C05456=1029.880,242.416,382.549,170.287,45.519,158.700
C05457=1029.874,242.168,382.577,170.284,45.520,158.700
C05458=1029.867,241.920,382.606,170.281,45.521,158.700
C05459=1029.860,241.672,382.634,170.277,45.522,158.700
C05460=1029.854,241.423,382.662,170.274,45.524,158.700
C05461=1029.847,241.175,382.691,170.271,45.524,158.699
C05462=1029.841,240.926,382.719,170.267,45.525,158.699
C05463=1029.834,240.678,382.748,170.264,45.527,158.699
C05464=1029.828,240.429,382.776,170.261,45.527,158.699
C05465=1029.821,240.181,382.805,170.259,45.529,158.699
C05466=1029.814,239.933,382.832,170.254,45.530,158.699
C05467=1029.808,239.685,382.861,170.252,45.531,158.699
C05468=1029.801,239.436,382.889,170.249,45.532,158.699
C05469=1029.794,239.189,382.918,170.245,45.533,158.699
C05470=1029.788,238.940,382.945,170.242,45.535,158.699
C05471=1029.781,238.692,382.974,170.239,45.535,158.698
C05472=1029.775,238.444,383.002,170.235,45.537,158.698
C05473=1029.768,238.195,383.030,170.232,45.538,158.698
C05474=1029.761,237.947,383.058,170.229,45.539,158.698
C05475=1029.754,237.698,383.087,170.225,45.540,158.698
C05476=1029.748,237.449,383.115,170.223,45.541,158.698
C05477=1029.741,237.202,383.143,170.220,45.543,158.698
C05478=1029.734,236.953,383.171,170.216,45.543,158.698
C05479=1029.727,236.705,383.199,170.213,45.545,158.698
C05480=1029.722,236.456,383.227,170.210,45.546,158.698
C05481=1029.715,236.208,383.255,170.207,45.547,158.698
C05482=1029.708,235.960,383.283,170.203,45.548,158.697
C05483=1029.701,235.711,383.311,170.200,45.549,158.697
C05484=1029.694,235.463,383.339,170.198,45.550,158.697
C05485=1029.687,235.215,383.367,170.194,45.552,158.697
C05486=1029.678,234.842,383.409,170.189,45.554,158.697
C05487=1029.668,234.468,383.450,170.184,45.556,158.697
C05488=1029.658,234.095,383.493,170.181,45.557,158.697
C05489=1029.649,233.721,383.535,170.176,45.559,158.697
C05490=1029.642,233.473,383.563,170.172,45.560,158.697
C05491=1029.635,233.225,383.591,170.169,45.561,158.697
C05492=1029.629,232.976,383.618,170.166,45.563,158.697
C05493=1029.622,232.728,383.646,170.163,45.563,158.696
C05494=1029.615,232.480,383.675,170.159,45.565,158.696
C05495=1029.608,232.231,383.702,170.157,45.566,158.696
C05496=1029.602,231.983,383.731,170.154,45.567,158.696
C05497=1029.596,231.734,383.758,170.151,45.568,158.696
C05498=1029.589,231.486,383.786,170.147,45.570,158.696
C05499=1029.582,231.237,383.814,170.144,45.571,158.696
C05500=1029.576,230.989,383.842,170.141,45.572,158.696
C05501=1029.570,230.741,383.869,170.138,45.573,158.696
C05502=1029.563,230.493,383.897,170.135,45.575,158.696
C05503=1029.556,230.244,383.924,170.132,45.576,158.696
C05504=1029.550,229.996,383.952,170.129,45.577,158.696
C05505=1029.543,229.747,383.980,170.126,45.578,158.696
C05506=1029.536,229.499,384.008,170.122,45.580,158.696
C05507=1029.530,229.250,384.035,170.120,45.581,158.696
C05508=1029.523,229.002,384.063,170.117,45.583,158.696
C05509=1029.516,228.754,384.091,170.114,45.583,158.695
C05510=1029.509,228.505,384.118,170.110,45.585,158.695
C05511=1029.503,228.257,384.146,170.107,45.586,158.695
C05512=1029.497,228.008,384.173,170.104,45.588,158.695
C05513=1029.490,227.760,384.201,170.102,45.589,158.695
C05514=1029.484,227.511,384.228,170.098,45.590,158.695
C05515=1029.477,227.263,384.256,170.095,45.591,158.695
C05516=1029.470,227.015,384.284,170.092,45.593,158.695
C05517=1029.463,226.766,384.311,170.089,45.594,158.695
C05518=1029.457,226.518,384.338,170.085,45.596,158.695
C05519=1029.450,226.270,384.365,170.083,45.597,158.695
C05520=1029.444,226.021,384.393,170.080,45.598,158.695
C05521=1029.436,225.773,384.420,170.077,45.600,158.695
C05522=1029.430,225.524,384.447,170.073,45.601,158.695
C05523=1029.423,225.276,384.475,170.071,45.603,158.695
C05524=1029.417,225.028,384.502,170.068,45.604,158.695
C05525=1029.410,224.779,384.529,170.065,45.605,158.695
C05526=1029.403,224.531,384.556,170.061,45.607,158.695
C05527=1029.397,224.282,384.584,170.059,45.608,158.695
C05528=1029.390,224.033,384.611,170.056,45.610,158.695
C05529=1029.383,223.785,384.638,170.053,45.611,158.695
C05530=1029.377,223.537,384.666,170.049,45.612,158.695
C05531=1029.370,223.288,384.693,170.046,45.614,158.695
C05532=1029.364,223.040,384.720,170.043,45.615,158.694
C05533=1029.356,222.792,384.748,170.041,45.616,158.694
C05534=1029.351,222.543,384.774,170.038,45.617,158.694
C05535=1029.344,222.295,384.802,170.034,45.619,158.694
C05536=1029.338,222.046,384.829,170.031,45.620,158.694
C05537=1029.330,221.798,384.856,170.029,45.621,158.694
C05538=1029.323,221.549,384.884,170.026,45.623,158.694
C05539=1029.318,221.301,384.910,170.023,45.624,158.694
C05540=1029.311,221.052,384.938,170.019,45.626,158.694
C05541=1029.304,220.804,384.965,170.016,45.627,158.694
C05542=1029.294,220.423,385.006,170.012,45.630,158.694
C05543=1029.284,220.042,385.049,170.007,45.631,158.694
C05544=1029.274,219.661,385.090,170.004,45.634,158.694
C05545=1029.264,219.279,385.131,169.999,45.636,158.694
C05546=1029.257,219.032,385.158,169.995,45.638,158.694
C05547=1029.251,218.783,385.185,169.993,45.639,158.694
C05548=1029.244,218.534,385.212,169.990,45.640,158.694
C05549=1029.237,218.286,385.239,169.987,45.642,158.694
C05550=1029.230,218.038,385.265,169.984,45.643,158.694
C05551=1029.224,217.789,385.293,169.980,45.645,158.694
C05552=1029.217,217.540,385.319,169.978,45.647,158.694
C05553=1029.211,217.292,385.346,169.975,45.648,158.694
C05554=1029.203,217.044,385.373,169.972,45.649,158.694
C05555=1029.197,216.795,385.400,169.970,45.651,158.694
C05556=1029.191,216.547,385.426,169.966,45.652,158.694
C05557=1029.183,216.298,385.453,169.963,45.654,158.694
C05558=1029.177,216.050,385.480,169.961,45.656,158.694
C05559=1029.170,215.802,385.507,169.958,45.657,158.694
C05560=1029.164,215.552,385.534,169.955,45.658,158.694
C05561=1029.156,215.304,385.561,169.951,45.660,158.694
C05562=1029.151,215.056,385.587,169.948,45.661,158.694
C05563=1029.144,214.807,385.614,169.946,45.663,158.694
C05564=1029.137,214.558,385.641,169.943,45.665,158.694
C05565=1029.131,214.310,385.667,169.940,45.666,158.694
C05566=1029.124,214.062,385.695,169.938,45.667,158.694
C05567=1029.117,213.813,385.721,169.934,45.669,158.694
C05568=1029.110,213.565,385.747,169.931,45.671,158.694
C05569=1029.104,213.316,385.774,169.929,45.672,158.694
C05570=1029.098,213.068,385.800,169.926,45.674,158.694
C05571=1029.091,212.819,385.828,169.923,45.675,158.694
C05572=1029.084,212.571,385.854,169.920,45.676,158.694
C05573=1029.078,212.322,385.881,169.917,45.679,158.694
C05574=1029.071,212.073,385.907,169.914,45.680,158.694
C05575=1029.065,211.825,385.934,169.911,45.681,158.694
C05576=1029.058,211.576,385.960,169.908,45.683,158.694
C05577=1029.051,211.328,385.987,169.906,45.685,158.695
C05578=1029.045,211.080,386.014,169.903,45.686,158.695
C05579=1029.038,210.831,386.041,169.900,45.687,158.695
C05580=1029.032,210.583,386.067,169.897,45.689,158.694
C05581=1029.025,210.334,386.094,169.894,45.691,158.695
C05582=1029.018,210.086,386.120,169.891,45.692,158.695
C05583=1029.011,209.837,386.146,169.889,45.694,158.695
C05584=1029.005,209.589,386.173,169.886,45.696,158.695
C05585=1028.998,209.340,386.199,169.883,45.697,158.695
C05586=1028.991,209.091,386.226,169.881,45.698,158.695
C05587=1028.985,208.843,386.252,169.877,45.701,158.695
C05588=1028.978,208.594,386.279,169.874,45.702,158.695
C05589=1028.972,208.346,386.305,169.872,45.703,158.695
C05590=1028.965,208.097,386.331,169.869,45.705,158.695
C05591=1028.958,207.849,386.357,169.866,45.707,158.695
C05592=1028.951,207.601,386.384,169.864,45.708,158.695
C05593=1028.946,207.352,386.410,169.861,45.710,158.695
C05594=1028.938,207.103,386.436,169.857,45.712,158.695
C05595=1028.932,206.855,386.462,169.855,45.714,158.695
C05596=1028.925,206.606,386.488,169.852,45.715,158.695
C05597=1028.918,206.358,386.514,169.849,45.716,158.695
C05598=1028.908,205.982,386.554,169.845,45.720,158.695
C05599=1028.899,205.606,386.594,169.840,45.722,158.695
C05600=1028.888,205.231,386.633,169.837,45.724,158.695
C05601=1028.878,204.855,386.673,169.832,45.727,158.695
C05602=1028.852,203.809,386.777,169.464,45.624,158.634
C05603=1028.846,203.560,386.802,169.460,45.626,158.634
C05604=1028.841,203.311,386.826,169.456,45.628,158.634
C05605=1028.835,203.063,386.851,169.452,45.631,158.634
C05606=1028.829,202.814,386.876,169.449,45.633,158.634
C05607=1028.822,202.566,386.900,169.444,45.636,158.634
C05608=1028.817,202.317,386.925,169.441,45.638,158.635
C05609=1028.811,202.069,386.950,169.437,45.641,158.635
C05610=1028.805,201.819,386.975,169.433,45.643,158.635
C05611=1028.799,201.570,386.999,169.430,45.646,158.635
C05612=1028.793,201.322,387.024,169.426,45.648,158.635
C05613=1028.787,201.073,387.048,169.423,45.650,158.635
C05614=1028.781,200.825,387.073,169.418,45.653,158.635
C05615=1028.775,200.576,387.098,169.415,45.656,158.635
C05616=1028.769,200.327,387.122,169.411,45.658,158.635
C05617=1028.763,200.078,387.146,169.407,45.660,158.635
C05618=1028.757,199.830,387.171,169.403,45.663,158.636
C05619=1028.751,199.581,387.195,169.400,45.666,158.636
C05620=1028.745,199.332,387.220,169.395,45.668,158.636
C05621=1028.739,199.083,387.244,169.392,45.671,158.636
C05622=1028.733,198.834,387.268,169.389,45.673,158.636
C05623=1028.727,198.585,387.292,169.384,45.676,158.636
C05624=1028.721,198.338,387.317,169.381,45.679,158.636
C05625=1028.714,198.089,387.341,169.377,45.682,158.637
C05626=1028.709,197.839,387.366,169.374,45.684,158.637
C05627=1028.703,197.591,387.389,169.370,45.687,158.637
C05628=1028.697,197.342,387.414,169.366,45.689,158.637
C05629=1028.691,197.093,387.438,169.363,45.692,158.637
C05630=1028.685,196.844,387.462,169.358,45.695,158.637
C05631=1028.679,196.596,387.486,169.355,45.697,158.637
C05632=1028.672,196.347,387.510,169.352,45.700,158.637
C05633=1028.667,196.098,387.534,169.348,45.703,158.638
C05634=1028.660,195.849,387.558,169.344,45.705,158.638
C05635=1028.655,195.601,387.582,169.340,45.707,158.638
C05636=1028.648,195.352,387.606,169.337,45.710,158.638
C05637=1028.643,195.103,387.631,169.333,45.712,158.638
C05638=1028.636,194.854,387.655,169.329,45.716,158.638
C05639=1028.631,194.606,387.679,169.326,45.718,158.638
C05640=1028.624,194.357,387.703,169.322,45.721,158.639
C05641=1028.619,194.108,387.727,169.319,45.723,158.639
C05642=1028.612,193.859,387.751,169.315,45.726,158.639
C05643=1028.606,193.611,387.775,169.311,45.729,158.639
C05644=1028.601,193.362,387.799,169.308,45.731,158.639
C05645=1028.594,193.113,387.823,169.305,45.734,158.639
C05646=1028.589,192.865,387.847,169.301,45.736,158.640
C05647=1028.582,192.616,387.871,169.297,45.740,158.640
C05648=1028.577,192.366,387.895,169.293,45.742,158.640
C05649=1028.571,192.117,387.919,169.290,45.745,158.640
C05650=1028.565,191.869,387.943,169.286,45.747,158.640
C05651=1028.559,191.621,387.967,169.283,45.750,158.640
C05652=1028.553,191.372,387.991,169.279,45.752,158.640
C05653=1028.548,191.123,388.015,169.275,45.755,158.641
C05654=1028.542,190.874,388.038,169.272,45.758,158.641
C05655=1028.536,190.625,388.063,169.269,45.760,158.641
C05656=1028.530,190.377,388.086,169.265,45.763,158.641
C05657=1028.523,190.128,388.111,169.261,45.766,158.641
C05658=1028.518,189.879,388.135,169.258,45.769,158.641
C05659=1028.512,189.630,388.158,169.254,45.771,158.641
C05660=1028.506,189.381,388.182,169.251,45.774,158.642
C05661=1028.500,189.133,388.206,169.247,45.776,158.642
C05662=1028.495,188.884,388.230,169.244,45.779,158.642
C05663=1028.488,188.600,388.257,169.240,45.782,158.642
C05664=1028.482,188.317,388.284,169.235,45.785,158.642
C05665=1028.474,188.034,388.311,169.232,45.788,158.643
C05666=1028.468,187.751,388.338,169.228,45.791,158.643
C05667=1028.463,187.502,388.362,169.224,45.794,158.643
C05668=1028.456,187.253,388.386,169.221,45.797,158.643
C05669=1028.450,187.005,388.410,169.218,45.799,158.643
C05670=1028.445,186.756,388.433,169.213,45.802,158.643
C05671=1028.439,186.507,388.457,169.210,45.804,158.643
C05672=1028.434,186.257,388.481,169.207,45.807,158.644
C05673=1028.428,186.009,388.504,169.203,45.810,158.644
C05674=1028.422,185.761,388.528,169.200,45.812,158.644
C05675=1028.417,185.512,388.552,169.197,45.815,158.644
C05676=1028.410,185.263,388.576,169.193,45.817,158.644
C05677=1028.405,185.014,388.599,169.190,45.820,158.644
C05678=1028.399,184.765,388.623,169.186,45.823,158.645
C05679=1028.393,184.517,388.647,169.183,45.826,158.645
C05680=1028.388,184.268,388.670,169.180,45.829,158.645
C05681=1028.381,184.019,388.694,169.176,45.831,158.645
C05682=1028.376,183.770,388.718,169.172,45.834,158.645
C05683=1028.370,183.521,388.741,169.168,45.836,158.645
C05684=1028.364,183.272,388.764,169.165,45.839,158.646
C05685=1028.359,183.024,388.789,169.162,45.842,158.646
C05686=1028.353,182.775,388.811,169.158,45.844,158.646
C05687=1028.347,182.526,388.835,169.155,45.847,158.646
C05688=1028.341,182.277,388.858,169.152,45.850,158.646
C05689=1028.335,182.028,388.881,169.149,45.853,158.647
C05690=1028.329,181.780,388.904,169.145,45.856,158.647
C05691=1028.323,181.530,388.927,169.141,45.859,158.647
C05692=1028.317,181.282,388.951,169.138,45.862,158.647
C05693=1028.311,181.033,388.974,169.135,45.865,158.647
C05694=1028.304,180.784,388.996,169.131,45.868,158.648
C05695=1028.298,180.535,389.019,169.128,45.871,158.648
C05696=1028.292,180.286,389.043,169.125,45.874,158.648
C05697=1028.286,180.037,389.066,169.121,45.876,158.648
C05698=1028.280,179.789,389.089,169.118,45.879,158.648
C05699=1028.274,179.540,389.111,169.114,45.882,158.649
C05700=1028.268,179.290,389.135,169.111,45.885,158.649
C05701=1028.262,179.041,389.157,169.107,45.888,158.649
C05702=1028.256,178.793,389.180,169.104,45.891,158.649
C05703=1028.250,178.544,389.204,169.101,45.894,158.650
C05704=1028.244,178.296,389.226,169.098,45.897,158.650
C05705=1028.238,178.047,389.249,169.094,45.900,158.650
C05706=1028.232,177.797,389.273,169.091,45.903,158.650
C05707=1028.226,177.548,389.296,169.088,45.906,158.650
C05708=1028.219,177.300,389.318,169.085,45.908,158.651
C05709=1028.214,177.051,389.341,169.080,45.912,158.651
C05710=1028.208,176.802,389.364,169.077,45.915,158.651
C05711=1028.202,176.553,389.387,169.074,45.917,158.651
C05712=1028.197,176.304,389.410,169.071,45.920,158.652
C05713=1028.190,176.056,389.432,169.067,45.923,158.652
C05714=1028.184,175.807,389.455,169.064,45.926,158.652
C05715=1028.178,175.557,389.478,169.061,45.929,158.652
C05716=1028.172,175.308,389.501,169.058,45.932,158.652
C05717=1028.166,175.060,389.524,169.054,45.934,158.653
C05718=1028.160,174.811,389.547,169.051,45.937,158.653
C05719=1028.154,174.562,389.570,169.048,45.940,158.653
C05720=1028.149,174.313,389.593,169.044,45.943,158.653
C05721=1028.142,174.064,389.615,169.041,45.946,158.653
C05722=1028.136,173.815,389.638,169.038,45.949,158.654
C05723=1028.131,173.566,389.661,169.035,45.952,158.654
C05724=1028.125,173.318,389.684,169.031,45.955,158.654
C05725=1028.118,173.069,389.706,169.028,45.958,158.654
C05726=1028.113,172.820,389.729,169.025,45.961,158.655
C05727=1028.106,172.536,389.755,169.021,45.965,158.655
C05728=1028.099,172.253,389.781,169.018,45.968,158.655
C05729=1028.093,171.969,389.807,169.013,45.971,158.655
C05730=1028.086,171.685,389.832,169.009,45.975,158.656
C05731=1028.080,171.436,389.855,169.006,45.978,158.656
C05732=1028.074,171.187,389.878,169.003,45.980,158.656
C05733=1028.068,170.939,389.901,169.001,45.983,158.656
C05734=1028.063,170.690,389.923,168.997,45.986,158.657
C05735=1028.057,170.441,389.945,168.994,45.989,158.657
C05736=1028.052,170.192,389.968,168.991,45.992,158.657
C05737=1028.045,169.943,389.991,168.988,45.995,158.657
C05738=1028.039,169.695,390.014,168.984,45.998,158.658
C05739=1028.034,169.446,390.037,168.981,46.001,158.658
C05740=1028.028,169.196,390.059,168.978,46.004,158.658
C05741=1028.022,168.948,390.081,168.975,46.007,158.658
C05742=1028.016,168.699,390.104,168.971,46.010,158.658
C05743=1028.010,168.450,390.127,168.968,46.013,158.659
C05744=1028.004,168.201,390.149,168.965,46.015,158.659
C05745=1027.998,167.952,390.172,168.961,46.018,158.659
C05746=1027.993,167.703,390.195,168.958,46.021,158.659
C05747=1027.987,167.454,390.218,168.955,46.024,158.659
C05748=1027.981,167.205,390.239,168.952,46.027,158.660
C05749=1027.976,166.956,390.262,168.948,46.030,158.660
C05750=1027.970,166.708,390.285,168.945,46.032,158.660
C05751=1027.964,166.458,390.307,168.942,46.035,158.660
C05752=1027.958,166.209,390.329,168.940,46.038,158.661
C05753=1027.952,165.961,390.352,168.936,46.041,158.661
C05754=1027.947,165.711,390.375,168.933,46.044,158.661
C05755=1027.941,165.463,390.396,168.930,46.047,158.661
C05756=1027.935,165.214,390.419,168.927,46.050,158.662
C05757=1027.930,164.965,390.442,168.923,46.053,158.662
C05758=1027.924,164.716,390.465,168.920,46.056,158.662
C05759=1027.918,164.467,390.486,168.917,46.059,158.662
C05760=1027.912,164.218,390.509,168.914,46.062,158.662
C05761=1027.907,163.970,390.532,168.911,46.064,158.663
C05762=1027.901,163.720,390.553,168.908,46.067,158.663
C05763=1027.895,163.471,390.576,168.905,46.070,158.663
C05764=1027.890,163.222,390.599,168.902,46.073,158.663
C05765=1027.884,162.973,390.622,168.898,46.076,158.664
C05766=1027.878,162.725,390.644,168.895,46.079,158.664
C05767=1027.873,162.476,390.666,168.892,46.082,158.664
C05768=1027.867,162.227,390.689,168.890,46.085,158.664
C05769=1027.861,161.978,390.710,168.887,46.088,158.665
C05770=1027.856,161.729,390.733,168.883,46.091,158.665
C05771=1027.850,161.480,390.755,168.880,46.094,158.665
C05772=1027.844,161.231,390.777,168.877,46.097,158.665
C05773=1027.838,160.982,390.800,168.874,46.100,158.665
C05774=1027.833,160.734,390.822,168.870,46.103,158.666
C05775=1027.828,160.484,390.845,168.868,46.105,158.666
C05776=1027.821,160.235,390.867,168.865,46.108,158.666
C05777=1027.816,159.986,390.889,168.862,46.111,158.666
C05778=1027.811,159.737,390.911,168.858,46.114,158.667
C05779=1027.805,159.488,390.933,168.855,46.117,158.667
C05780=1027.799,159.239,390.956,168.853,46.120,158.667
C05781=1027.793,158.990,390.977,168.850,46.123,158.668
C05782=1027.787,158.742,390.999,168.847,46.126,158.668
C05783=1027.782,158.492,391.021,168.843,46.129,158.668
C05784=1027.776,158.243,391.043,168.840,46.132,158.668
C05785=1027.769,157.994,391.065,168.837,46.135,158.668
C05786=1027.764,157.746,391.087,168.834,46.139,158.669
C05787=1027.758,157.497,391.109,168.831,46.142,158.669
C05788=1027.752,157.247,391.131,168.827,46.145,158.669
C05789=1027.746,156.998,391.152,168.825,46.147,158.670
C05790=1027.740,156.750,391.173,168.822,46.151,158.670
C05791=1027.733,156.465,391.199,168.818,46.154,158.670
C05792=1027.726,156.182,391.224,168.815,46.158,158.670
C05793=1027.720,155.897,391.248,168.811,46.162,158.671
C05794=1027.713,155.614,391.273,168.808,46.165,158.671
C05795=1027.708,155.364,391.295,168.805,46.168,158.671
C05796=1027.702,155.115,391.317,168.802,46.171,158.672
C05797=1027.696,154.866,391.339,168.799,46.174,158.672
C05798=1027.690,154.618,391.361,168.796,46.177,158.672
C05799=1027.684,154.369,391.383,168.793,46.180,158.672
C05800=1027.678,154.119,391.405,168.790,46.184,158.673
C05801=1027.673,153.871,391.426,168.787,46.187,158.673
C05802=1027.666,153.622,391.447,168.784,46.190,158.673
C05803=1027.661,153.372,391.470,168.780,46.192,158.673
C05804=1027.655,153.124,391.491,168.778,46.196,158.674
C05805=1027.649,152.874,391.513,168.775,46.199,158.674
C05806=1027.643,152.625,391.534,168.772,46.202,158.674
C05807=1027.638,152.377,391.555,168.769,46.205,158.675
C05808=1027.631,152.128,391.577,168.766,46.208,158.675
C05809=1027.625,151.878,391.599,168.762,46.211,158.675
C05810=1027.620,151.630,391.620,168.760,46.214,158.675
C05811=1027.613,151.381,391.642,168.757,46.218,158.676
C05812=1027.607,151.131,391.663,168.754,46.221,158.676
C05813=1027.603,150.883,391.685,168.751,46.224,158.676
C05814=1027.596,150.633,391.707,168.748,46.227,158.677
C05815=1027.591,150.385,391.728,168.745,46.230,158.677
C05816=1027.585,150.136,391.750,168.742,46.233,158.677
C05817=1027.578,149.887,391.771,168.739,46.236,158.677
C05818=1027.573,149.637,391.792,168.736,46.240,158.678
C05819=1027.567,149.388,391.813,168.733,46.243,158.678
C05820=1027.561,149.140,391.835,168.730,46.246,158.678
C05821=1027.555,148.890,391.856,168.728,46.249,158.679
C05822=1027.549,148.641,391.878,168.724,46.252,158.679
C05823=1027.544,148.393,391.899,168.721,46.255,158.679
C05824=1027.537,148.144,391.921,168.718,46.258,158.679
C05825=1027.532,147.895,391.942,168.715,46.261,158.680
C05826=1027.526,147.645,391.963,168.713,46.264,158.680
C05827=1027.520,147.397,391.984,168.710,46.267,158.680
C05828=1027.514,147.148,392.006,168.707,46.271,158.681
C05829=1027.508,146.898,392.028,168.703,46.274,158.681
C05830=1027.503,146.650,392.049,168.700,46.277,158.681
C05831=1027.497,146.400,392.070,168.698,46.280,158.681
C05832=1027.491,146.151,392.091,168.695,46.283,158.682
C05833=1027.485,145.902,392.113,168.692,46.286,158.682
C05834=1027.480,145.653,392.133,168.689,46.290,158.682
C05835=1027.474,145.404,392.155,168.686,46.293,158.682
C05836=1027.468,145.155,392.176,168.684,46.296,158.683
C05837=1027.461,144.906,392.197,168.680,46.299,158.683
C05838=1027.455,144.657,392.218,168.677,46.303,158.683
C05839=1027.450,144.408,392.239,168.674,46.306,158.684
C05840=1027.444,144.158,392.260,168.671,46.309,158.684
C05841=1027.438,143.910,392.282,168.669,46.312,158.684
C05842=1027.432,143.661,392.303,168.666,46.315,158.685
C05843=1027.426,143.412,392.323,168.663,46.319,158.685
C05844=1027.420,143.163,392.345,168.660,46.322,158.685
C05845=1027.414,142.914,392.366,168.657,46.324,158.685
C05846=1027.409,142.664,392.387,168.654,46.328,158.686
C05847=1027.403,142.416,392.408,168.651,46.331,158.686
C05848=1027.396,142.166,392.429,168.648,46.335,158.686
C05849=1027.391,141.918,392.450,168.646,46.337,158.687
C05850=1027.385,141.668,392.471,168.643,46.340,158.687
C05851=1027.379,141.419,392.492,168.640,46.344,158.687
C05852=1027.373,141.170,392.514,168.637,46.347,158.688
C05853=1027.368,140.921,392.534,168.633,46.350,158.688
C05854=1027.362,140.673,392.555,168.631,46.353,158.688
C05855=1027.355,140.388,392.579,168.627,46.357,158.688
C05856=1027.349,140.103,392.603,168.625,46.361,158.689
C05857=1027.342,139.819,392.627,168.621,46.364,158.689
C05858=1027.335,139.535,392.651,168.618,46.368,158.689
C05859=1027.330,139.286,392.672,168.615,46.371,158.690
C05860=1027.323,139.037,392.693,168.612,46.374,158.690
C05861=1027.318,138.788,392.713,168.609,46.377,158.690
C05862=1027.312,138.539,392.735,168.607,46.381,158.691
C05863=1027.306,138.290,392.755,168.604,46.384,158.691
C05864=1027.300,138.040,392.776,168.601,46.387,158.691
C05865=1027.294,137.792,392.797,168.598,46.390,158.692
C05866=1027.288,137.543,392.817,168.596,46.394,158.692
C05867=1027.282,137.294,392.839,168.592,46.397,158.692
C05868=1027.277,137.044,392.859,168.589,46.400,158.693
C05869=1027.270,136.795,392.880,168.587,46.403,158.693
C05870=1027.265,136.546,392.901,168.584,46.407,158.693
C05871=1027.259,136.297,392.921,168.581,46.410,158.693
C05872=1027.253,136.048,392.942,168.578,46.413,158.694
C05873=1027.247,135.799,392.963,168.576,46.416,158.694
C05874=1027.241,135.550,392.983,168.573,46.420,158.694
C05875=1027.235,135.301,393.004,168.570,46.423,158.695
C05876=1027.229,135.052,393.025,168.567,46.426,158.695
C05877=1027.223,134.803,393.046,168.565,46.429,158.695
C05878=1027.217,134.554,393.065,168.561,46.432,158.696
C05879=1027.211,134.304,393.086,168.558,46.436,158.696
C05880=1027.206,134.056,393.108,168.555,46.439,158.696
C05881=1027.200,133.807,393.128,168.553,46.442,158.697
C05882=1027.194,133.557,393.149,168.550,46.445,158.697
C05883=1027.188,133.308,393.169,168.547,46.449,158.697
C05884=1027.182,133.060,393.190,168.545,46.452,158.697
C05885=1027.176,132.810,393.210,168.542,46.455,158.698
C05886=1027.171,132.561,393.231,168.539,46.458,158.698
C05887=1027.165,132.312,393.251,168.536,46.462,158.698
C05888=1027.159,132.062,393.272,168.534,46.465,158.699
C05889=1027.152,131.814,393.292,168.531,46.468,158.699
C05890=1027.147,131.565,393.313,168.527,46.471,158.699
C05891=1027.141,131.315,393.334,168.525,46.475,158.700
C05892=1027.135,131.066,393.354,168.522,46.478,158.700
C05893=1027.130,130.817,393.374,168.519,46.482,158.700
C05894=1027.124,130.568,393.394,168.517,46.484,158.701
C05895=1027.118,130.319,393.415,168.514,46.488,158.701
C05896=1027.112,130.070,393.436,168.511,46.491,158.701
C05897=1027.106,129.822,393.456,168.508,46.495,158.702
C05898=1027.099,129.572,393.476,168.506,46.497,158.702
C05899=1027.093,129.323,393.496,168.503,46.501,158.702
C05900=1027.088,129.074,393.517,168.500,46.505,158.703
C05901=1027.082,128.825,393.537,168.497,46.508,158.703
C05902=1027.076,128.575,393.556,168.495,46.511,158.703
C05903=1027.070,128.326,393.576,168.492,46.515,158.704
C05904=1027.063,128.077,393.596,168.489,46.518,158.704
C05905=1027.058,127.828,393.617,168.486,46.521,158.704
C05906=1027.052,127.579,393.637,168.484,46.525,158.705
C05907=1027.045,127.329,393.657,168.480,46.528,158.705
C05908=1027.039,127.081,393.677,168.478,46.532,158.705
C05909=1027.034,126.831,393.698,168.475,46.534,158.705
C05910=1027.028,126.583,393.718,168.472,46.538,158.706
C05911=1027.022,126.333,393.738,168.469,46.542,158.706
C05912=1027.016,126.084,393.758,168.466,46.545,158.706
C05913=1027.010,125.835,393.778,168.464,46.548,158.707
C05914=1027.004,125.587,393.798,168.461,46.552,158.707
C05915=1026.998,125.336,393.818,168.458,46.555,158.707
C05916=1026.992,125.087,393.838,168.456,46.558,158.708
C05917=1026.986,124.839,393.858,168.453,46.561,158.708
C05918=1026.980,124.590,393.878,168.450,46.565,158.708
C05919=1026.974,124.305,393.901,168.447,46.569,158.709
C05920=1026.966,124.021,393.924,168.444,46.572,158.709
C05921=1026.959,123.736,393.947,168.441,46.576,158.710
C05922=1026.953,123.452,393.970,168.437,46.580,158.710
C05923=1026.947,123.203,393.990,168.435,46.583,158.710
C05924=1026.941,122.954,394.010,168.432,46.587,158.711
C05925=1026.935,122.704,394.029,168.429,46.590,158.711
C05926=1026.929,122.455,394.050,168.427,46.593,158.711
C05927=1026.923,122.206,394.070,168.424,46.596,158.712
C05928=1026.917,121.957,394.090,168.421,46.600,158.712
C05929=1026.911,121.708,394.110,168.419,46.603,158.712
C05930=1026.906,121.459,394.129,168.416,46.607,158.713
C05931=1026.900,121.209,394.150,168.413,46.610,158.713
C05932=1026.894,120.960,394.170,168.411,46.613,158.713
C05933=1026.888,120.711,394.190,168.408,46.617,158.714
C05934=1026.882,120.462,394.209,168.405,46.620,158.714
C05935=1026.876,120.213,394.229,168.403,46.623,158.714
C05936=1026.870,119.964,394.249,168.400,46.626,158.714
C05937=1026.864,119.715,394.270,168.398,46.630,158.715
C05938=1026.859,119.465,394.289,168.395,46.633,158.715
C05939=1026.853,119.216,394.309,168.391,46.636,158.715
C05940=1026.847,118.968,394.329,168.390,46.640,158.716
C05941=1026.841,118.718,394.348,168.386,46.643,158.716
C05942=1026.835,118.469,394.368,168.383,46.647,158.716
C05943=1026.830,118.220,394.389,168.381,46.649,158.717
C05944=1026.824,117.971,394.408,168.378,46.653,158.717
C05945=1026.818,117.722,394.428,168.375,46.656,158.717
C05946=1026.811,117.472,394.449,168.373,46.659,158.718
C05947=1026.806,117.223,394.468,168.370,46.663,158.718
C05948=1026.800,116.974,394.488,168.368,46.666,158.718
C05949=1026.795,116.725,394.508,168.365,46.670,158.719
C05950=1026.789,116.476,394.528,168.362,46.673,158.719
C05951=1026.783,116.227,394.547,168.360,46.676,158.719
C05952=1026.777,115.978,394.567,168.357,46.679,158.720
C05953=1026.771,115.729,394.587,168.355,46.683,158.720
C05954=1026.765,115.480,394.607,168.352,46.686,158.720
C05955=1026.759,115.230,394.626,168.349,46.689,158.721
C05956=1026.754,114.981,394.646,168.346,46.692,158.721
C05957=1026.749,114.732,394.666,168.344,46.696,158.721
C05958=1026.743,114.483,394.686,168.341,46.698,158.722
C05959=1026.737,114.234,394.706,168.338,46.702,158.722
C05960=1026.731,113.985,394.725,168.336,46.705,158.722
C05961=1026.725,113.736,394.745,168.333,46.709,158.723
C05962=1026.720,113.486,394.765,168.330,46.712,158.723
C05963=1026.713,113.237,394.785,168.328,46.715,158.723
C05964=1026.708,112.987,394.804,168.325,46.718,158.723
C05965=1026.702,112.738,394.824,168.323,46.722,158.724
C05966=1026.696,112.489,394.843,168.320,46.725,158.724
C05967=1026.690,112.240,394.863,168.317,46.728,158.724
C05968=1026.684,111.991,394.883,168.315,46.732,158.725
C05969=1026.678,111.742,394.901,168.312,46.735,158.725
C05970=1026.672,111.493,394.921,168.309,46.738,158.725
C05971=1026.666,111.243,394.940,168.307,46.742,158.726
C05972=1026.660,110.995,394.960,168.304,46.745,158.726
C05973=1026.654,110.745,394.980,168.302,46.748,158.727
C05974=1026.649,110.496,394.999,168.299,46.752,158.727
C05975=1026.643,110.247,395.019,168.296,46.755,158.727
C05976=1026.637,109.997,395.038,168.294,46.759,158.728
C05977=1026.631,109.748,395.057,168.291,46.762,158.728
C05978=1026.625,109.499,395.077,168.288,46.765,158.728
C05979=1026.619,109.250,395.096,168.286,46.769,158.729
C05980=1026.613,109.001,395.115,168.283,46.772,158.729
C05981=1026.607,108.751,395.134,168.281,46.775,158.729
C05982=1026.601,108.503,395.154,168.278,46.779,158.730
C05983=1026.594,108.218,395.176,168.275,46.783,158.730
C05984=1026.588,107.933,395.197,168.272,46.787,158.730
C05985=1026.580,107.649,395.219,168.268,46.791,158.731
C05986=1026.573,107.364,395.241,168.265,46.795,158.731
C05987=1026.567,107.115,395.261,168.263,46.798,158.732
C05988=1026.562,106.865,395.280,168.260,46.801,158.732
C05989=1026.555,106.616,395.299,168.257,46.805,158.732
C05990=1026.550,106.367,395.318,168.255,46.808,158.733
C05991=1026.544,106.118,395.338,168.252,46.811,158.733
C05992=1026.537,105.869,395.356,168.250,46.815,158.733
C05993=1026.532,105.620,395.375,168.247,46.819,158.734
C05994=1026.526,105.371,395.395,168.244,46.822,158.734
C05995=1026.520,105.122,395.413,168.242,46.825,158.734
C05996=1026.514,104.872,395.432,168.239,46.829,158.735
C05997=1026.508,104.623,395.452,168.237,46.832,158.735
C05998=1026.503,104.374,395.472,168.234,46.835,158.735
C05999=1026.496,104.125,395.490,168.231,46.839,158.736
C06000=1026.490,103.875,395.510,168.229,46.842,158.736
C06001=1026.485,103.626,395.529,168.226,46.846,158.736
C06002=1026.478,103.377,395.547,168.224,46.849,158.737
C06003=1026.473,103.127,395.567,168.221,46.852,158.737
C06004=1026.467,102.878,395.586,168.218,46.856,158.737
C06005=1026.461,102.629,395.605,168.216,46.859,158.738
C06006=1026.455,102.381,395.624,168.213,46.862,158.738
C06007=1026.449,102.131,395.643,168.211,46.866,158.738
C06008=1026.443,101.882,395.662,168.208,46.869,158.739
C06009=1026.437,101.633,395.681,168.206,46.872,158.739
C06010=1026.432,101.383,395.701,168.203,46.876,158.739
C06011=1026.425,101.134,395.719,168.200,46.879,158.739
C06012=1026.420,100.885,395.738,168.198,46.882,158.740
C06013=1026.414,100.636,395.757,168.195,46.886,158.740
C06014=1026.408,100.387,395.776,168.193,46.889,158.741
C06015=1026.402,100.138,395.795,168.190,46.893,158.741
C06016=1026.397,99.888,395.814,168.188,46.896,158.741
C06017=1026.390,99.639,395.833,168.185,46.899,158.742
C06018=1026.385,99.390,395.852,168.182,46.903,158.742
C06019=1026.378,99.140,395.871,168.180,46.906,158.742
C06020=1026.372,98.891,395.890,168.177,46.910,158.743
C06021=1026.366,98.641,395.908,168.175,46.913,158.743
C06022=1026.361,98.393,395.926,168.172,46.917,158.743
C06023=1026.355,98.143,395.946,168.169,46.920,158.744
C06024=1026.348,97.894,395.964,168.167,46.924,158.744
C06025=1026.342,97.645,395.983,168.164,46.927,158.744
C06026=1026.336,97.396,396.002,168.161,46.931,158.745
C06027=1026.330,97.147,396.021,168.159,46.934,158.745
C06028=1026.325,96.897,396.039,168.156,46.937,158.745
C06029=1026.319,96.648,396.058,168.154,46.941,158.746
C06030=1026.312,96.399,396.076,168.151,46.944,158.746
C06031=1026.307,96.150,396.096,168.148,46.948,158.746
C06032=1026.300,95.900,396.114,168.146,46.951,158.747
C06033=1026.294,95.651,396.133,168.143,46.955,158.747
C06034=1026.289,95.402,396.151,168.141,46.958,158.748
C06035=1026.282,95.153,396.170,168.138,46.962,158.748
C06036=1026.277,94.903,396.189,168.135,46.965,158.748
C06037=1026.270,94.654,396.208,168.133,46.968,158.749
C06038=1026.264,94.405,396.226,168.130,46.972,158.749
C06039=1026.259,94.156,396.244,168.128,46.975,158.749
C06040=1026.253,93.907,396.263,168.125,46.979,158.750
C06041=1026.247,93.657,396.282,168.123,46.982,158.750
C06042=1026.241,93.408,396.300,168.120,46.985,158.750
C06043=1026.235,93.159,396.319,168.117,46.989,158.750
C06044=1026.229,92.910,396.338,168.115,46.992,158.751
C06045=1026.223,92.661,396.356,168.112,46.996,158.751
C06046=1026.217,92.411,396.374,168.110,46.999,158.752
C06047=1026.211,92.127,396.396,168.107,47.003,158.752
C06048=1026.204,91.843,396.417,168.105,47.007,158.752
C06049=1026.197,91.557,396.438,168.102,47.011,158.753
C06050=1026.190,91.273,396.459,168.099,47.014,158.753
C06051=1026.184,91.024,396.478,168.096,47.018,158.754
C06052=1026.179,90.775,396.497,168.093,47.021,158.754
C06053=1026.172,90.525,396.515,168.091,47.025,158.754
C06054=1026.167,90.276,396.534,168.088,47.028,158.755
C06055=1026.161,90.026,396.552,168.086,47.031,158.755
C06056=1026.155,89.778,396.570,168.083,47.035,158.755
C06057=1026.149,89.528,396.589,168.081,47.039,158.756
C06058=1026.143,89.279,396.607,168.078,47.042,158.756
C06059=1026.137,89.030,396.626,168.075,47.045,158.756
C06060=1026.131,88.781,396.644,168.073,47.049,158.757
C06061=1026.125,88.531,396.662,168.070,47.053,158.757
C06062=1026.119,88.282,396.680,168.068,47.056,158.757
C06063=1026.113,88.033,396.698,168.065,47.059,158.758
C06064=1026.107,87.783,396.716,168.062,47.063,158.758
C06065=1026.100,87.534,396.735,168.060,47.066,158.758
C06066=1026.094,87.285,396.753,168.057,47.070,158.759
C06067=1026.089,87.036,396.772,168.055,47.074,158.759
C06068=1026.083,86.786,396.790,168.052,47.077,158.759
C06069=1026.076,86.537,396.808,168.049,47.080,158.760
C06070=1026.071,86.288,396.826,168.047,47.084,158.760
C06071=1026.064,86.039,396.845,168.045,47.088,158.760
C06072=1026.058,85.789,396.863,168.042,47.090,158.761
C06073=1026.053,85.540,396.880,168.039,47.094,158.761
C06074=1026.046,85.291,396.899,168.037,47.098,158.761
C06075=1026.040,85.041,396.917,168.035,47.101,158.762
C06076=1026.034,84.793,396.935,168.031,47.104,158.762
C06077=1026.028,84.543,396.953,168.030,47.108,158.762
C06078=1026.022,84.293,396.971,168.027,47.112,158.763
C06079=1026.016,84.045,396.989,168.025,47.115,158.763
C06080=1026.010,83.795,397.007,168.022,47.118,158.763
C06081=1026.004,83.546,397.026,168.019,47.122,158.764
C06082=1025.998,83.297,397.043,168.017,47.125,158.764
C06083=1025.992,83.047,397.061,168.014,47.129,158.765
C06084=1025.987,82.798,397.080,168.012,47.132,158.765
C06085=1025.981,82.549,397.098,168.009,47.136,158.765
C06086=1025.975,82.299,397.116,168.007,47.139,158.766
C06087=1025.969,82.051,397.134,168.004,47.143,158.766
C06088=1025.963,81.801,397.152,168.001,47.146,158.766
C06089=1025.957,81.551,397.170,167.999,47.150,158.767
C06090=1025.951,81.303,397.188,167.996,47.153,158.767
C06091=1025.945,81.053,397.206,167.994,47.156,158.767
C06092=1025.939,80.804,397.224,167.991,47.160,158.768
C06093=1025.933,80.555,397.243,167.989,47.163,158.768
C06094=1025.927,80.305,397.260,167.986,47.166,158.768
C06095=1025.921,80.056,397.278,167.984,47.170,158.769
C06096=1025.915,79.807,397.297,167.981,47.174,158.769
C06097=1025.909,79.558,397.314,167.978,47.178,158.769
C06098=1025.903,79.308,397.332,167.976,47.180,158.770
C06099=1025.898,79.059,397.350,167.973,47.184,158.770
C06100=1025.891,78.810,397.368,167.971,47.188,158.770
C06101=1025.885,78.560,397.386,167.968,47.191,158.771
C06102=1025.880,78.311,397.404,167.966,47.194,158.771
C06103=1025.874,78.061,397.422,167.963,47.198,158.771
C06104=1025.868,77.813,397.440,167.961,47.201,158.772
C06105=1025.862,77.563,397.458,167.958,47.204,158.772
C06106=1025.856,77.314,397.476,167.956,47.208,158.772
C06107=1025.850,77.064,397.494,167.953,47.211,158.773
C06108=1025.844,76.815,397.511,167.950,47.215,158.773
C06109=1025.838,76.566,397.529,167.948,47.218,158.773
C06110=1025.832,76.316,397.547,167.946,47.222,158.774
C06111=1025.825,76.032,397.567,167.943,47.226,158.774
C06112=1025.818,75.747,397.587,167.940,47.230,158.774
C06113=1025.811,75.463,397.607,167.937,47.234,158.775
C06114=1025.805,75.178,397.628,167.934,47.238,158.775
C06115=1025.799,74.929,397.645,167.931,47.242,158.776
C06116=1025.792,74.679,397.662,167.929,47.244,158.776
C06117=1025.787,74.430,397.680,167.926,47.248,158.776
C06118=1025.780,74.181,397.699,167.924,47.252,158.777
C06119=1025.775,73.932,397.716,167.922,47.255,158.777
C06120=1025.768,73.683,397.734,167.919,47.259,158.777
C06121=1025.763,73.434,397.751,167.917,47.262,158.778
C06122=1025.756,73.184,397.769,167.914,47.266,158.778
C06123=1025.751,72.935,397.787,167.912,47.269,158.779
C06124=1025.744,72.686,397.804,167.909,47.273,158.779
C06125=1025.739,72.437,397.822,167.907,47.276,158.779
C06126=1025.732,72.187,397.840,167.904,47.280,158.779
C06127=1025.727,71.938,397.857,167.902,47.283,158.780
C06128=1025.720,71.688,397.874,167.899,47.287,158.780
C06129=1025.715,71.439,397.892,167.896,47.290,158.780
C06130=1025.709,71.189,397.909,167.894,47.294,158.781
C06131=1025.703,70.940,397.927,167.891,47.297,158.781
C06132=1025.696,70.690,397.944,167.889,47.300,158.781
C06133=1025.691,70.441,397.962,167.886,47.304,158.782
C06134=1025.685,70.192,397.980,167.884,47.307,158.782
C06135=1025.678,69.943,397.997,167.881,47.311,158.783
C06136=1025.673,69.694,398.014,167.878,47.314,158.783
C06137=1025.667,69.444,398.032,167.876,47.318,158.783
C06138=1025.661,69.195,398.049,167.873,47.322,158.784
C06139=1025.654,68.946,398.067,167.871,47.325,158.784
C06140=1025.649,68.697,398.085,167.868,47.328,158.784
C06141=1025.642,68.447,398.101,167.866,47.332,158.785
C06142=1025.637,68.198,398.119,167.864,47.335,158.785
C06143=1025.631,67.948,398.137,167.862,47.339,158.785
C06144=1025.624,67.699,398.154,167.858,47.342,158.786
C06145=1025.619,67.450,398.171,167.856,47.346,158.786
C06146=1025.612,67.200,398.188,167.854,47.349,158.786
C06147=1025.607,66.951,398.205,167.851,47.353,158.787
C06148=1025.600,66.702,398.223,167.849,47.356,158.787
C06149=1025.594,66.452,398.240,167.846,47.360,158.787
C06150=1025.589,66.203,398.258,167.843,47.364,158.788
C06151=1025.582,65.953,398.274,167.841,47.367,158.788
C06152=1025.577,65.704,398.292,167.838,47.370,158.788
C06153=1025.570,65.455,398.309,167.836,47.374,158.789
C06154=1025.565,65.205,398.326,167.833,47.377,158.789
C06155=1025.559,64.957,398.343,167.831,47.381,158.789
C06156=1025.552,64.707,398.361,167.828,47.385,158.790
C06157=1025.546,64.458,398.378,167.825,47.388,158.790
C06158=1025.540,64.208,398.395,167.823,47.391,158.790
C06159=1025.534,63.959,398.412,167.820,47.395,158.791
C06160=1025.529,63.710,398.430,167.819,47.399,158.791
C06161=1025.522,63.460,398.447,167.815,47.402,158.791
C06162=1025.517,63.211,398.464,167.814,47.405,158.792
C06163=1025.510,62.961,398.481,167.811,47.409,158.792
C06164=1025.504,62.712,398.498,167.808,47.413,158.793
C06165=1025.498,62.463,398.515,167.806,47.416,158.793
C06166=1025.492,62.213,398.532,167.803,47.420,158.793
C06167=1025.485,61.964,398.549,167.800,47.424,158.794
C06168=1025.479,61.715,398.565,167.798,47.427,158.794
C06169=1025.473,61.465,398.582,167.795,47.431,158.794
C06170=1025.467,61.216,398.599,167.792,47.434,158.795
C06171=1025.461,60.966,398.617,167.790,47.438,158.795
C06172=1025.455,60.717,398.633,167.787,47.442,158.795
C06173=1025.448,60.468,398.650,167.785,47.445,158.796
C06174=1025.442,60.218,398.667,167.783,47.449,158.796
C06175=1025.436,59.977,398.683,167.780,47.453,158.796
C06176=1025.430,59.735,398.700,167.778,47.456,158.797
C06177=1025.425,59.492,398.716,167.775,47.459,158.797
C06178=1025.419,59.251,398.732,167.773,47.463,158.798
C06179=1025.413,59.009,398.748,167.770,47.467,158.798
C06180=1025.407,58.767,398.765,167.768,47.470,158.798
C06181=1025.401,58.526,398.780,167.765,47.473,158.798
C06182=1025.395,58.284,398.797,167.763,47.477,158.799
C06183=1025.389,58.035,398.814,167.760,47.481,158.799
C06184=1025.382,57.785,398.831,167.757,47.484,158.800
C06185=1025.377,57.535,398.848,167.755,47.487,158.800
C06186=1025.371,57.286,398.865,167.752,47.491,158.800
C06187=1025.364,57.036,398.881,167.751,47.495,158.801
C06188=1025.358,56.788,398.898,167.748,47.498,158.801
C06189=1025.352,56.538,398.914,167.745,47.502,158.801
C06190=1025.347,56.289,398.931,167.743,47.505,158.802
C06191=1025.340,56.039,398.949,167.740,47.509,158.802
C06192=1025.334,55.790,398.965,167.738,47.512,158.802
C06193=1025.328,55.541,398.982,167.735,47.516,158.803
C06194=1025.321,55.291,398.999,167.732,47.520,158.803
C06195=1025.316,55.041,399.015,167.730,47.523,158.803
C06196=1025.310,54.793,399.032,167.727,47.527,158.804
C06197=1025.304,54.543,399.049,167.725,47.530,158.804
C06198=1025.298,54.294,399.065,167.722,47.534,158.804
C06199=1025.291,54.045,399.082,167.719,47.538,158.805
C06200=1025.286,53.795,399.099,167.717,47.541,158.805
C06201=1025.280,53.546,399.115,167.714,47.544,158.805
C06202=1025.273,53.297,399.132,167.713,47.548,158.806
C06203=1025.267,53.047,399.149,167.710,47.552,158.806
C06204=1025.261,52.797,399.165,167.707,47.555,158.806
C06205=1025.255,52.548,399.181,167.705,47.558,158.807
C06206=1025.249,52.299,399.199,167.702,47.562,158.807
C06207=1025.242,51.999,399.219,167.699,47.566,158.807
C06208=1025.235,51.700,399.239,167.696,47.571,158.808
C06209=1025.227,51.400,399.258,167.692,47.575,158.808
C06210=1025.220,51.100,399.278,167.690,47.579,158.809
C06211=1025.215,50.851,399.296,167.687,47.583,158.809
C06212=1025.208,50.601,399.312,167.685,47.586,158.809
C06213=1025.202,50.351,399.328,167.682,47.590,158.810
C06214=1025.196,50.102,399.345,167.680,47.593,158.810
C06215=1025.190,49.853,399.362,167.677,47.597,158.810
C06216=1025.184,49.604,399.378,167.674,47.600,158.811
C06217=1025.179,49.354,399.395,167.672,47.604,158.811
C06218=1025.172,49.104,399.411,167.669,47.607,158.811
C06219=1025.166,48.855,399.428,167.667,47.610,158.812
C06220=1025.160,48.606,399.445,167.664,47.614,158.812
C06221=1025.154,48.357,399.461,167.663,47.618,158.812
C06222=1025.149,48.107,399.478,167.659,47.621,158.813
C06223=1025.143,47.858,399.494,167.656,47.625,158.813
C06224=1025.137,47.608,399.510,167.655,47.628,158.813
C06225=1025.131,47.359,399.526,167.651,47.631,158.813
C06226=1025.124,47.110,399.544,167.650,47.635,158.814
C06227=1025.118,46.860,399.560,167.647,47.639,158.814
C06228=1025.113,46.611,399.577,167.645,47.641,158.814
C06229=1025.107,46.361,399.593,167.642,47.645,158.815
C06230=1025.101,46.112,399.609,167.640,47.649,158.815
C06231=1025.095,45.863,399.626,167.637,47.652,158.815
C06232=1025.089,45.613,399.642,167.634,47.656,158.816
C06233=1025.083,45.365,399.659,167.632,47.659,158.816
C06234=1025.077,45.115,399.675,167.629,47.662,158.816
C06235=1025.072,44.866,399.692,167.627,47.666,158.817
C06236=1025.066,44.616,399.708,167.624,47.669,158.817
C06237=1025.060,44.367,399.725,167.622,47.673,158.817
C06238=1025.054,44.118,399.741,167.619,47.676,158.818
C06239=1025.047,43.833,399.760,167.616,47.680,158.818
C06240=1025.040,43.547,399.778,167.613,47.684,158.818
C06241=1025.034,43.262,399.798,167.611,47.688,158.819
C06242=1025.027,42.976,399.816,167.608,47.692,158.819
C06243=1025.021,42.727,399.832,167.605,47.695,158.819
C06244=1025.015,42.478,399.848,167.603,47.698,158.820
C06245=1025.009,42.228,399.865,167.600,47.702,158.820
C06246=1025.003,41.979,399.881,167.598,47.706,158.820
C06247=1024.997,41.730,399.897,167.595,47.710,158.821
C06248=1024.990,41.481,399.913,167.592,47.713,158.821
C06249=1024.984,41.231,399.929,167.590,47.716,158.821
C06250=1024.979,40.982,399.945,167.587,47.720,158.822
C06251=1024.973,40.733,399.962,167.585,47.724,158.822
C06252=1024.967,40.483,399.978,167.582,47.727,158.822
C06253=1024.961,40.233,399.993,167.579,47.731,158.823
C06254=1024.955,39.984,400.010,167.577,47.734,158.823
C06255=1024.949,39.735,400.026,167.574,47.737,158.823
C06256=1024.942,39.485,400.042,167.572,47.741,158.824
C06257=1024.936,39.236,400.058,167.570,47.745,158.824
C06258=1024.930,38.987,400.074,167.567,47.748,158.824
C06259=1024.925,38.737,400.090,167.565,47.751,158.825
C06260=1024.919,38.487,400.106,167.562,47.755,158.825
C06261=1024.913,38.238,400.122,167.559,47.759,158.825
C06262=1024.907,37.989,400.138,167.557,47.762,158.825
C06263=1024.901,37.739,400.155,167.554,47.766,158.826
C06264=1024.894,37.490,400.170,167.552,47.769,158.826
C06265=1024.889,37.240,400.186,167.549,47.772,158.826
C06266=1024.883,36.991,400.202,167.547,47.776,158.827
C06267=1024.877,36.742,400.218,167.544,47.780,158.827
C06268=1024.871,36.492,400.235,167.541,47.784,158.828
C06269=1024.864,36.243,400.250,167.539,47.786,158.828
C06270=1024.858,35.993,400.266,167.536,47.790,158.828
C06271=1024.852,35.744,400.281,167.533,47.794,158.828
C06272=1024.846,35.494,400.297,167.532,47.798,158.829
C06273=1024.840,35.245,400.313,167.529,47.802,158.829
C06274=1024.834,34.995,400.328,167.526,47.805,158.829
C06275=1024.828,34.746,400.344,167.524,47.808,158.830
C06276=1024.822,34.497,400.361,167.521,47.812,158.830
C06277=1024.816,34.247,400.376,167.518,47.816,158.830
C06278=1024.810,33.998,400.392,167.516,47.819,158.831
C06279=1024.804,33.749,400.407,167.513,47.823,158.831
C06280=1024.798,33.499,400.423,167.510,47.826,158.831
C06281=1024.792,33.250,400.439,167.508,47.830,158.832
C06282=1024.786,33.000,400.454,167.506,47.834,158.832
C06283=1024.780,32.751,400.470,167.502,47.837,158.832
C06284=1024.774,32.502,400.487,167.501,47.841,158.833
C06285=1024.767,32.252,400.501,167.498,47.844,158.833
C06286=1024.761,32.003,400.518,167.496,47.847,158.833
C06287=1024.755,31.753,400.533,167.493,47.851,158.834
C06288=1024.749,31.504,400.549,167.490,47.855,158.834
C06289=1024.743,31.254,400.564,167.488,47.858,158.834
C06290=1024.737,31.005,400.580,167.485,47.862,158.835
C06291=1024.732,30.755,400.595,167.482,47.865,158.835
C06292=1024.725,30.506,400.611,167.480,47.869,158.835
C06293=1024.719,30.257,400.627,167.477,47.873,158.836
C06294=1024.713,30.007,400.643,167.474,47.876,158.836
C06295=1024.707,29.758,400.658,167.472,47.880,158.836
C06296=1024.701,29.508,400.674,167.469,47.883,158.837
C06297=1024.695,29.259,400.690,167.467,47.886,158.837
C06298=1024.689,29.010,400.705,167.464,47.890,158.837
C06299=1024.683,28.760,400.721,167.462,47.894,158.837
C06300=1024.677,28.511,400.736,167.459,47.897,158.838
C06301=1024.671,28.261,400.752,167.457,47.901,158.838
C06302=1024.665,28.011,400.768,167.454,47.905,158.838
C06303=1024.658,27.727,400.785,167.451,47.908,158.839
C06304=1024.651,27.442,400.803,167.448,47.912,158.839
C06305=1024.645,27.157,400.821,167.446,47.917,158.840
C06306=1024.637,26.871,400.838,167.443,47.921,158.840
C06307=1024.631,26.622,400.854,167.440,47.924,158.840
C06308=1024.626,26.373,400.868,167.437,47.928,158.840
C06309=1024.619,26.124,400.884,167.435,47.931,158.841
C06310=1024.613,25.874,400.900,167.432,47.935,158.841
C06311=1024.607,25.624,400.915,167.429,47.939,158.841
C06312=1024.601,25.374,400.930,167.427,47.942,158.842
C06313=1024.595,25.125,400.946,167.424,47.946,158.842
C06314=1024.589,24.876,400.960,167.421,47.950,158.842
C06315=1024.583,24.626,400.976,167.419,47.953,158.843
C06316=1024.576,24.377,400.992,167.416,47.956,158.843
C06317=1024.570,24.127,401.007,167.413,47.960,158.843
C06318=1024.564,23.877,401.022,167.411,47.964,158.844
C06319=1024.559,23.628,401.037,167.409,47.968,158.844
C06320=1024.553,23.379,401.053,167.406,47.971,158.844
C06321=1024.546,23.129,401.068,167.403,47.975,158.845
C06322=1024.540,22.880,401.083,167.401,47.978,158.845
C06323=1024.535,22.631,401.098,167.398,47.982,158.845
C06324=1024.528,22.382,401.114,167.395,47.985,158.845
C06325=1024.522,22.132,401.129,167.393,47.989,158.846
C06326=1024.516,21.882,401.144,167.390,47.993,158.846
C06327=1024.510,21.633,401.159,167.387,47.996,158.846
C06328=1024.504,21.383,401.174,167.385,47.999,158.847
C06329=1024.498,21.134,401.190,167.382,48.003,158.847
C06330=1024.492,20.884,401.205,167.380,48.007,158.847
C06331=1024.486,20.635,401.219,167.377,48.010,158.848
C06332=1024.480,20.385,401.235,167.375,48.014,158.848
C06333=1024.474,20.136,401.250,167.372,48.018,158.848
C06334=1024.469,19.886,401.265,167.370,48.021,158.849
C06335=1024.462,19.637,401.281,167.367,48.024,158.849
C06336=1024.456,19.388,401.296,167.364,48.028,158.849
C06337=1024.449,19.138,401.311,167.362,48.031,158.849
C06338=1024.444,18.889,401.326,167.359,48.035,158.850
C06339=1024.438,18.639,401.341,167.356,48.039,158.850
C06340=1024.432,18.389,401.356,167.354,48.042,158.851
C06341=1024.426,18.141,401.370,167.351,48.046,158.851
C06342=1024.420,17.891,401.386,167.348,48.049,158.851
C06343=1024.414,17.641,401.401,167.345,48.053,158.851
C06344=1024.407,17.391,401.416,167.344,48.057,158.852
C06345=1024.402,17.142,401.430,167.341,48.060,158.852
C06346=1024.395,16.893,401.445,167.338,48.064,158.852
C06347=1024.390,16.643,401.461,167.336,48.068,158.853
C06348=1024.384,16.394,401.475,167.333,48.071,158.853
C06349=1024.377,16.144,401.490,167.330,48.075,158.853
C06350=1024.371,15.894,401.505,167.328,48.078,158.854
C06351=1024.365,15.645,401.520,167.325,48.082,158.854
C06352=1024.360,15.395,401.535,167.322,48.085,158.854
C06353=1024.354,15.147,401.550,167.319,48.089,158.854
C06354=1024.347,14.897,401.565,167.317,48.093,158.855
C06355=1024.341,14.647,401.580,167.314,48.096,158.855
C06356=1024.335,14.398,401.594,167.311,48.100,158.855
C06357=1024.329,14.149,401.609,167.310,48.103,158.856
C06358=1024.323,13.899,401.625,167.306,48.106,158.856
C06359=1024.317,13.650,401.640,167.304,48.110,158.856
C06360=1024.311,13.400,401.654,167.302,48.114,158.857
C06361=1024.305,13.150,401.669,167.299,48.118,158.857
C06362=1024.299,12.901,401.683,167.296,48.121,158.857
C06363=1024.293,12.651,401.698,167.293,48.125,158.857
C06364=1024.287,12.402,401.713,167.291,48.128,158.858
C06365=1024.281,12.153,401.728,167.288,48.132,158.858
C06366=1024.274,11.903,401.742,167.285,48.136,158.858
C06367=1024.267,11.619,401.759,167.283,48.140,158.859
C06368=1024.260,11.336,401.775,167.279,48.144,158.859
C06369=1024.253,11.052,401.792,167.276,48.149,158.860
C06370=1024.247,10.769,401.809,167.273,48.153,158.860
C06371=1024.240,10.519,401.822,167.271,48.156,158.860
C06372=1024.234,10.270,401.837,167.268,48.160,158.860
C06373=1024.228,10.020,401.852,167.266,48.163,158.861
C06374=1024.221,9.770,401.867,167.263,48.167,158.861
C06375=1024.216,9.521,401.881,167.260,48.171,158.861
C06376=1024.210,9.271,401.896,167.257,48.175,158.862
C06377=1024.204,9.022,401.910,167.254,48.179,158.862
C06378=1024.198,8.772,401.924,167.252,48.182,158.862
C06379=1024.192,8.523,401.939,167.249,48.186,158.863
C06380=1024.185,8.273,401.954,167.246,48.189,158.863
C06381=1024.180,8.024,401.969,167.244,48.193,158.863
C06382=1024.173,7.774,401.982,167.242,48.196,158.863
C06383=1024.166,7.525,401.997,167.239,48.200,158.864
C06384=1024.161,7.276,402.012,167.236,48.204,158.864
C06385=1024.155,7.026,402.026,167.233,48.208,158.864
C06386=1024.149,6.777,402.041,167.231,48.211,158.865
C06387=1024.143,6.526,402.055,167.228,48.215,158.865
C06388=1024.137,6.277,402.069,167.225,48.218,158.865
C06389=1024.131,6.028,402.084,167.222,48.222,158.865
C06390=1024.125,5.778,402.098,167.220,48.225,158.866
C06391=1024.119,5.528,402.113,167.217,48.229,158.866
C06392=1024.112,5.280,402.127,167.215,48.233,158.867
C06393=1024.106,5.030,402.141,167.211,48.236,158.867
C06394=1024.100,4.781,402.156,167.210,48.240,158.867
C06395=1024.094,4.530,402.170,167.207,48.244,158.867
C06396=1024.089,4.281,402.185,167.204,48.247,158.868
C06397=1024.083,4.032,402.199,167.201,48.251,158.868
C06398=1024.077,3.782,402.214,167.199,48.254,158.868
C06399=1024.071,3.533,402.228,167.196,48.258,158.868
C06400=1024.065,3.283,402.242,167.193,48.261,158.869
C06401=1024.058,3.034,402.256,167.190,48.265,158.869
C06402=1024.052,2.784,402.271,167.188,48.268,158.869
C06403=1024.046,2.535,402.285,167.185,48.272,158.870
C06404=1024.040,2.285,402.299,167.182,48.276,158.870
C06405=1024.035,2.036,402.314,167.179,48.279,158.870
C06406=1024.029,1.786,402.328,167.177,48.283,158.871
C06407=1024.023,1.537,402.343,167.175,48.287,158.871
C06408=1024.017,1.287,402.357,167.172,48.290,158.871
C06409=1024.010,1.038,402.371,167.169,48.294,158.871
C06410=1024.005,0.788,402.385,167.167,48.297,158.872
C06411=1023.999,0.539,402.399,167.164,48.301,158.872
C06412=1023.993,0.289,402.414,167.161,48.305,158.872
C06413=1023.987,0.040,402.428,167.158,48.308,158.872
C06414=1023.981,-0.210,402.442,167.156,48.311,158.873
C06415=1023.975,-0.460,402.456,167.153,48.315,158.873
C06416=1023.970,-0.709,402.471,167.150,48.318,158.873
C06417=1023.963,-0.959,402.485,167.148,48.322,158.874
C06418=1023.957,-1.208,402.499,167.145,48.325,158.874
C06419=1023.952,-1.457,402.513,167.142,48.329,158.874
C06420=1023.945,-1.708,402.527,167.139,48.332,158.874
C06421=1023.940,-1.957,402.542,167.137,48.336,158.875
C06422=1023.934,-2.206,402.556,167.134,48.339,158.875
C06423=1023.928,-2.456,402.571,167.131,48.343,158.875
C06424=1023.922,-2.706,402.584,167.128,48.347,158.875
C06425=1023.916,-2.955,402.598,167.126,48.350,158.876
C06426=1023.910,-3.204,402.613,167.124,48.354,158.876
C06427=1023.904,-3.454,402.627,167.120,48.357,158.876
C06428=1023.898,-3.704,402.641,167.119,48.361,158.877
C06429=1023.892,-3.953,402.655,167.115,48.364,158.877
C06430=1023.887,-4.203,402.669,167.113,48.368,158.877
C06431=1023.880,-4.485,402.685,167.110,48.372,158.877
C06432=1023.873,-4.766,402.700,167.106,48.376,158.878
C06433=1023.866,-5.048,402.715,167.103,48.380,158.878
C06434=1023.859,-5.330,402.731,167.101,48.384,158.878
C06435=1023.853,-5.579,402.745,167.098,48.388,158.879
C06436=1023.847,-5.829,402.759,167.095,48.391,158.879
C06437=1023.841,-6.079,402.773,167.092,48.395,158.879
C06438=1023.835,-6.328,402.786,167.089,48.399,158.879
C06439=1023.829,-6.577,402.801,167.086,48.403,158.880
C06440=1023.822,-6.827,402.814,167.084,48.406,158.880
C06441=1023.817,-7.077,402.828,167.081,48.410,158.880
C06442=1023.810,-7.326,402.841,167.078,48.414,158.881
C06443=1023.804,-7.576,402.856,167.076,48.418,158.881
C06444=1023.798,-7.826,402.869,167.072,48.421,158.881
C06445=1023.793,-8.075,402.883,167.070,48.425,158.881
C06446=1023.786,-8.324,402.896,167.068,48.428,158.882
C06447=1023.780,-8.575,402.910,167.065,48.432,158.882
C06448=1023.774,-8.824,402.924,167.062,48.435,158.882
C06449=1023.768,-9.073,402.938,167.059,48.439,158.883
C06450=1023.762,-9.322,402.951,167.056,48.443,158.883
C06451=1023.756,-9.572,402.966,167.054,48.446,158.883
C06452=1023.750,-9.822,402.979,167.051,48.450,158.883
C06453=1023.744,-10.071,402.993,167.049,48.454,158.884
C06454=1023.738,-10.321,403.006,167.045,48.457,158.884
C06455=1023.733,-10.570,403.020,167.043,48.461,158.884
C06456=1023.726,-10.820,403.034,167.040,48.465,158.885
C06457=1023.720,-11.070,403.047,167.038,48.468,158.885
C06458=1023.714,-11.319,403.061,167.035,48.472,158.885
C06459=1023.709,-11.569,403.075,167.032,48.475,158.885
C06460=1023.702,-11.818,403.088,167.029,48.479,158.886
C06461=1023.696,-12.068,403.102,167.026,48.483,158.886
C06462=1023.690,-12.317,403.115,167.023,48.486,158.886
C06463=1023.685,-12.567,403.129,167.021,48.490,158.886
C06464=1023.679,-12.816,403.142,167.018,48.494,158.887
C06465=1023.673,-13.066,403.156,167.015,48.497,158.887
C06466=1023.666,-13.316,403.170,167.012,48.501,158.887
C06467=1023.661,-13.566,403.183,167.009,48.504,158.887
C06468=1023.655,-13.815,403.196,167.007,48.508,158.888
C06469=1023.649,-14.065,403.210,167.005,48.512,158.888
C06470=1023.643,-14.314,403.224,167.001,48.515,158.888
C06471=1023.637,-14.563,403.237,166.999,48.519,158.889
C06472=1023.631,-14.813,403.251,166.996,48.522,158.889
C06473=1023.625,-15.063,403.264,166.993,48.526,158.889
C06474=1023.619,-15.312,403.278,166.991,48.529,158.889
C06475=1023.613,-15.562,403.291,166.988,48.533,158.890
C06476=1023.608,-15.812,403.305,166.985,48.537,158.890
C06477=1023.602,-16.061,403.318,166.982,48.541,158.890
C06478=1023.595,-16.310,403.331,166.979,48.544,158.890
C06479=1023.589,-16.560,403.344,166.976,48.548,158.891
C06480=1023.584,-16.810,403.358,166.973,48.552,158.891
C06481=1023.577,-17.060,403.371,166.972,48.555,158.891
C06482=1023.571,-17.309,403.384,166.968,48.558,158.891
C06483=1023.565,-17.558,403.398,166.966,48.562,158.892
C06484=1023.560,-17.809,403.411,166.963,48.566,158.892
C06485=1023.553,-18.058,403.424,166.960,48.570,158.892
C06486=1023.547,-18.307,403.437,166.957,48.573,158.893
C06487=1023.541,-18.557,403.450,166.954,48.577,158.893
C06488=1023.535,-18.806,403.463,166.951,48.581,158.893
C06489=1023.530,-19.056,403.477,166.948,48.585,158.893
C06490=1023.523,-19.305,403.490,166.946,48.588,158.894
C06491=1023.517,-19.555,403.503,166.944,48.592,158.894
C06492=1023.511,-19.805,403.517,166.940,48.595,158.894
C06493=1023.505,-20.055,403.529,166.938,48.599,158.894
C06494=1023.499,-20.304,403.543,166.935,48.603,158.895
C06495=1023.493,-20.584,403.557,166.932,48.607,158.895
C06496=1023.486,-20.864,403.572,166.928,48.611,158.895
C06497=1023.479,-21.144,403.587,166.925,48.615,158.896
C06498=1023.472,-21.424,403.602,166.923,48.619,158.896
C06499=1023.466,-21.674,403.615,166.920,48.623,158.896
C06500=1023.460,-21.923,403.628,166.917,48.626,158.896
C06501=1023.454,-22.173,403.641,166.914,48.630,158.897
C06502=1023.448,-22.423,403.654,166.911,48.634,158.897
C06503=1023.443,-22.673,403.667,166.908,48.637,158.897
C06504=1023.437,-22.922,403.680,166.905,48.641,158.897
C06505=1023.430,-23.171,403.694,166.902,48.645,158.898
C06506=1023.425,-23.421,403.706,166.899,48.648,158.898
C06507=1023.418,-23.670,403.719,166.897,48.652,158.898
C06508=1023.412,-23.920,403.732,166.895,48.656,158.899
C06509=1023.407,-24.170,403.746,166.891,48.659,158.899
C06510=1023.401,-24.420,403.758,166.889,48.663,158.899
C06511=1023.395,-24.669,403.772,166.885,48.666,158.899
C06512=1023.389,-24.919,403.784,166.883,48.670,158.899
C06513=1023.383,-25.168,403.798,166.880,48.674,158.900
C06514=1023.377,-25.417,403.810,166.877,48.678,158.900
C06515=1023.372,-25.667,403.824,166.875,48.681,158.900
C06516=1023.366,-25.917,403.836,166.872,48.684,158.900
C06517=1023.360,-26.166,403.849,166.869,48.688,158.901
C06518=1023.354,-26.416,403.862,166.866,48.692,158.901
C06519=1023.348,-26.665,403.875,166.863,48.696,158.901
C06520=1023.342,-26.915,403.888,166.860,48.699,158.901
C06521=1023.337,-27.165,403.901,166.857,48.703,158.902
C06522=1023.330,-27.415,403.914,166.854,48.707,158.902
C06523=1023.324,-27.664,403.927,166.852,48.710,158.902
C06524=1023.318,-27.914,403.940,166.849,48.714,158.902
C06525=1023.312,-28.164,403.953,166.847,48.717,158.903
C06526=1023.307,-28.413,403.965,166.844,48.721,158.903
C06527=1023.300,-28.662,403.977,166.841,48.725,158.903
C06528=1023.294,-28.912,403.990,166.838,48.729,158.903
C06529=1023.288,-29.162,404.003,166.835,48.733,158.904
C06530=1023.282,-29.411,404.015,166.832,48.736,158.904
C06531=1023.276,-29.661,404.028,166.829,48.740,158.904
C06532=1023.270,-29.911,404.041,166.826,48.744,158.905
C06533=1023.264,-30.160,404.053,166.824,48.748,158.905
C06534=1023.258,-30.410,404.066,166.820,48.751,158.905
C06535=1023.253,-30.660,404.078,166.818,48.755,158.905
C06536=1023.247,-30.909,404.091,166.815,48.759,158.906
C06537=1023.240,-31.158,404.103,166.812,48.762,158.906
C06538=1023.234,-31.408,404.116,166.809,48.766,158.906
C06539=1023.228,-31.658,404.129,166.806,48.770,158.906
C06540=1023.222,-31.907,404.142,166.803,48.773,158.906
C06541=1023.216,-32.157,404.154,166.800,48.777,158.907
C06542=1023.211,-32.406,404.167,166.797,48.781,158.907
C06543=1023.205,-32.656,404.179,166.794,48.784,158.907
C06544=1023.199,-32.906,404.192,166.791,48.788,158.907
C06545=1023.193,-33.156,404.204,166.790,48.792,158.908
C06546=1023.186,-33.405,404.217,166.787,48.795,158.908
C06547=1023.181,-33.654,404.229,166.784,48.799,158.908
C06548=1023.175,-33.904,404.242,166.781,48.803,158.909
C06549=1023.169,-34.154,404.254,166.778,48.806,158.909
C06550=1023.163,-34.404,404.267,166.775,48.810,158.909
C06551=1023.157,-34.654,404.279,166.772,48.813,158.909
C06552=1023.152,-34.903,404.291,166.769,48.817,158.909
C06553=1023.146,-35.153,404.304,166.766,48.821,158.910
C06554=1023.140,-35.402,404.316,166.763,48.825,158.910
C06555=1023.133,-35.652,404.329,166.760,48.828,158.910
C06556=1023.128,-35.901,404.341,166.757,48.832,158.910
C06557=1023.122,-36.151,404.354,166.754,48.836,158.911
C06558=1023.116,-36.401,404.367,166.752,48.840,158.911
C06559=1023.109,-36.680,404.380,166.749,48.844,158.911
C06560=1023.103,-36.959,404.394,166.745,48.848,158.911
C06561=1023.097,-37.238,404.408,166.742,48.852,158.912
C06562=1023.090,-37.517,404.422,166.739,48.856,158.912
C06563=1023.084,-37.767,404.434,166.736,48.859,158.912
C06564=1023.079,-38.016,404.447,166.733,48.863,158.912
C06565=1023.073,-38.266,404.459,166.730,48.866,158.913
C06566=1023.067,-38.515,404.471,166.728,48.870,158.913
C06567=1023.061,-38.765,404.484,166.724,48.873,158.913
C06568=1023.055,-39.015,404.496,166.722,48.877,158.913
C06569=1023.049,-39.265,404.508,166.719,48.881,158.914
C06570=1023.044,-39.515,404.520,166.716,48.885,158.914
C06571=1023.037,-39.764,404.532,166.713,48.889,158.914
C06572=1023.031,-40.014,404.544,166.710,48.892,158.914
C06573=1023.026,-40.263,404.557,166.707,48.896,158.915
C06574=1023.019,-40.513,404.569,166.704,48.900,158.915
C06575=1023.013,-40.763,404.581,166.701,48.904,158.915
C06576=1023.008,-41.012,404.592,166.699,48.908,158.915
C06577=1023.002,-41.262,404.605,166.696,48.911,158.915
C06578=1022.996,-41.512,404.617,166.693,48.915,158.916
C06579=1022.990,-41.761,404.629,166.690,48.919,158.916
C06580=1022.984,-42.011,404.641,166.687,48.922,158.916
C06581=1022.978,-42.261,404.653,166.684,48.926,158.916
C06582=1022.972,-42.510,404.665,166.681,48.930,158.917
C06583=1022.966,-42.760,404.677,166.678,48.934,158.917
C06584=1022.960,-43.010,404.689,166.675,48.937,158.917
C06585=1022.954,-43.259,404.701,166.673,48.941,158.917
C06586=1022.948,-43.509,404.713,166.670,48.945,158.918
C06587=1022.943,-43.758,404.725,166.667,48.948,158.918
C06588=1022.937,-44.008,404.737,166.664,48.952,158.918
C06589=1022.931,-44.258,404.749,166.661,48.956,158.918
C06590=1022.925,-44.507,404.761,166.658,48.960,158.919
C06591=1022.919,-44.757,404.773,166.655,48.964,158.919
C06592=1022.913,-45.006,404.785,166.652,48.967,158.919
C06593=1022.907,-45.256,404.796,166.649,48.971,158.919
C06594=1022.901,-45.506,404.809,166.646,48.975,158.920
C06595=1022.896,-45.755,404.821,166.643,48.978,158.920
C06596=1022.889,-46.006,404.832,166.641,48.982,158.920
C06597=1022.884,-46.255,404.844,166.638,48.986,158.920
C06598=1022.877,-46.504,404.856,166.635,48.989,158.920
C06599=1022.872,-46.754,404.868,166.632,48.993,158.921
C06600=1022.866,-47.004,404.880,166.629,48.996,158.921
C06601=1022.860,-47.253,404.892,166.626,49.000,158.921
C06602=1022.855,-47.503,404.904,166.623,49.004,158.921
C06603=1022.849,-47.752,404.915,166.620,49.008,158.922
C06604=1022.843,-48.003,404.927,166.617,49.012,158.922
C06605=1022.837,-48.252,404.939,166.614,49.015,158.922
C06606=1022.831,-48.502,404.951,166.611,49.019,158.922
C06607=1022.826,-48.751,404.962,166.608,49.022,158.922
C06608=1022.820,-49.001,404.975,166.605,49.026,158.923
C06609=1022.815,-49.251,404.986,166.603,49.030,158.923
C06610=1022.808,-49.500,404.998,166.599,49.033,158.923
C06611=1022.803,-49.750,405.010,166.597,49.037,158.923
C06612=1022.796,-50.000,405.022,166.594,49.041,158.924
C06613=1022.791,-50.249,405.033,166.591,49.045,158.924
C06614=1022.785,-50.499,405.045,166.588,49.048,158.924
C06615=1022.780,-50.749,405.057,166.585,49.052,158.924
C06616=1022.773,-50.998,405.069,166.582,49.056,158.925
C06617=1022.767,-51.248,405.079,166.579,49.059,158.925
C06618=1022.761,-51.498,405.092,166.576,49.063,158.925
C06619=1022.756,-51.747,405.103,166.572,49.067,158.925
C06620=1022.749,-51.997,405.114,166.570,49.071,158.925
C06621=1022.743,-52.246,405.126,166.567,49.075,158.926
C06622=1022.737,-52.496,405.137,166.564,49.079,158.926
C06623=1022.731,-52.775,405.150,166.560,49.083,158.926
C06624=1022.724,-53.056,405.162,166.557,49.087,158.926
C06625=1022.718,-53.335,405.175,166.554,49.092,158.927
C06626=1022.711,-53.614,405.188,166.551,49.096,158.927
C06627=1022.704,-53.865,405.199,166.547,49.100,158.927
C06628=1022.699,-54.114,405.210,166.544,49.104,158.927
C06629=1022.693,-54.363,405.222,166.541,49.108,158.928
C06630=1022.687,-54.613,405.233,166.539,49.112,158.928
C06631=1022.681,-54.863,405.244,166.536,49.115,158.928
C06632=1022.675,-55.113,405.256,166.533,49.119,158.928
C06633=1022.669,-55.362,405.267,166.530,49.123,158.929
C06634=1022.663,-55.612,405.278,166.527,49.127,158.929
C06635=1022.657,-55.862,405.289,166.524,49.130,158.929
C06636=1022.652,-56.112,405.301,166.520,49.135,158.929
C06637=1022.646,-56.361,405.312,166.518,49.139,158.930
C06638=1022.639,-56.611,405.324,166.515,49.143,158.930
C06639=1022.634,-56.860,405.334,166.512,49.146,158.930
C06640=1022.627,-57.110,405.346,166.509,49.150,158.930
C06641=1022.622,-57.360,405.357,166.506,49.154,158.931
C06642=1022.616,-57.609,405.367,166.503,49.158,158.931
C06643=1022.610,-57.860,405.379,166.500,49.161,158.931
C06644=1022.604,-58.109,405.391,166.497,49.165,158.931
C06645=1022.599,-58.358,405.402,166.494,49.169,158.931
C06646=1022.592,-58.608,405.413,166.491,49.173,158.932
C06647=1022.586,-58.858,405.424,166.488,49.177,158.932
C06648=1022.581,-59.107,405.435,166.485,49.181,158.932
C06649=1022.576,-59.357,405.446,166.482,49.185,158.932
C06650=1022.569,-59.607,405.457,166.479,49.188,158.933
C06651=1022.564,-59.857,405.468,166.476,49.192,158.933
C06652=1022.558,-60.106,405.479,166.474,49.196,158.933
C06653=1022.552,-60.356,405.490,166.470,49.199,158.933
C06654=1022.546,-60.605,405.502,166.468,49.203,158.934
C06655=1022.540,-60.855,405.513,166.464,49.208,158.934
C06656=1022.534,-61.104,405.524,166.461,49.211,158.934
C06657=1022.528,-61.355,405.536,166.458,49.215,158.934
C06658=1022.523,-61.604,405.547,166.455,49.219,158.934
C06659=1022.517,-61.854,405.557,166.452,49.222,158.934
C06660=1022.511,-62.103,405.568,166.449,49.226,158.935
C06661=1022.505,-62.353,405.580,166.446,49.230,158.935
C06662=1022.499,-62.603,405.590,166.443,49.233,158.935
C06663=1022.493,-62.852,405.601,166.441,49.237,158.935
C06664=1022.488,-63.102,405.612,166.438,49.241,158.936
C06665=1022.483,-63.352,405.624,166.435,49.245,158.936
C06666=1022.476,-63.602,405.635,166.431,49.249,158.936
C06667=1022.471,-63.851,405.646,166.428,49.252,158.936
C06668=1022.465,-64.101,405.657,166.425,49.256,158.936
C06669=1022.459,-64.350,405.668,166.422,49.260,158.937
C06670=1022.454,-64.600,405.678,166.419,49.264,158.937
C06671=1022.447,-64.851,405.689,166.416,49.268,158.937
C06672=1022.442,-65.100,405.700,166.413,49.271,158.937
C06673=1022.437,-65.350,405.711,166.410,49.275,158.937
C06674=1022.431,-65.599,405.722,166.408,49.279,158.938
C06675=1022.425,-65.849,405.733,166.405,49.282,158.938
C06676=1022.419,-66.098,405.744,166.402,49.286,158.938
C06677=1022.414,-66.348,405.755,166.399,49.289,158.938
C06678=1022.407,-66.598,405.766,166.395,49.294,158.938
C06679=1022.402,-66.848,405.777,166.392,49.298,158.939
C06680=1022.396,-67.098,405.787,166.389,49.301,158.939
C06681=1022.390,-67.347,405.798,166.386,49.305,158.939
C06682=1022.385,-67.597,405.809,166.383,49.308,158.939
C06683=1022.380,-67.847,405.820,166.380,49.312,158.940
C06684=1022.374,-68.096,405.831,166.377,49.316,158.940
C06685=1022.368,-68.345,405.842,166.375,49.320,158.940
C06686=1022.363,-68.596,405.852,166.371,49.323,158.940
C06687=1022.356,-68.876,405.865,166.368,49.327,158.940
C06688=1022.349,-69.158,405.877,166.365,49.331,158.940
C06689=1022.343,-69.438,405.889,166.361,49.336,158.941
C06690=1022.337,-69.719,405.901,166.358,49.340,158.941
C06691=1022.331,-69.969,405.912,166.355,49.344,158.941
C06692=1022.326,-70.218,405.923,166.351,49.347,158.941
C06693=1022.320,-70.468,405.934,166.349,49.351,158.941
C06694=1022.314,-70.718,405.944,166.345,49.355,158.942
C06695=1022.309,-70.967,405.955,166.343,49.359,158.942
C06696=1022.303,-71.217,405.966,166.340,49.363,158.942
C06697=1022.297,-71.466,405.977,166.337,49.366,158.942
C06698=1022.292,-71.716,405.987,166.334,49.370,158.943
C06699=1022.286,-71.966,405.998,166.331,49.373,158.943
C06700=1022.280,-72.215,406.009,166.328,49.377,158.943
C06701=1022.275,-72.465,406.019,166.325,49.380,158.943
C06702=1022.269,-72.715,406.030,166.322,49.384,158.943
C06703=1022.264,-72.965,406.041,166.319,49.388,158.943
C06704=1022.259,-73.215,406.051,166.316,49.391,158.944
C06705=1022.253,-73.464,406.062,166.313,49.395,158.944
C06706=1022.247,-73.714,406.073,166.310,49.398,158.944
C06707=1022.242,-73.964,406.083,166.307,49.402,158.944
C06708=1022.236,-74.213,406.094,166.304,49.406,158.944
C06709=1022.231,-74.463,406.104,166.302,49.410,158.945
C06710=1022.225,-74.713,406.115,166.298,49.414,158.945
C06711=1022.219,-74.963,406.125,166.295,49.417,158.945
C06712=1022.213,-75.212,406.136,166.292,49.421,158.945
C06713=1022.208,-75.462,406.146,166.289,49.425,158.945
C06714=1022.202,-75.712,406.157,166.286,49.429,158.945
C06715=1022.196,-75.962,406.167,166.283,49.433,158.946
C06716=1022.190,-76.211,406.177,166.279,49.437,158.946
C06717=1022.185,-76.461,406.187,166.276,49.440,158.946
C06718=1022.179,-76.710,406.198,166.274,49.444,158.946
C06719=1022.174,-76.960,406.208,166.271,49.448,158.946
C06720=1022.168,-77.210,406.217,166.268,49.452,158.947
C06721=1022.162,-77.459,406.228,166.265,49.456,158.947
C06722=1022.157,-77.710,406.239,166.262,49.459,158.947
C06723=1022.151,-77.959,406.249,166.259,49.463,158.947
C06724=1022.145,-78.209,406.260,166.255,49.467,158.948
C06725=1022.139,-78.459,406.269,166.252,49.471,158.948
C06726=1022.133,-78.708,406.280,166.249,49.475,158.948
C06727=1022.129,-78.958,406.290,166.246,49.478,158.948
C06728=1022.123,-79.207,406.301,166.244,49.482,158.948
C06729=1022.117,-79.457,406.310,166.241,49.486,158.949
C06730=1022.111,-79.707,406.320,166.238,49.489,158.949
C06731=1022.106,-79.957,406.331,166.234,49.494,158.949
C06732=1022.100,-80.207,406.341,166.231,49.498,158.949
C06733=1022.094,-80.457,406.351,166.228,49.501,158.949
C06734=1022.089,-80.707,406.361,166.225,49.505,158.949
C06735=1022.083,-80.956,406.370,166.223,49.509,158.950
C06736=1022.077,-81.205,406.381,166.219,49.513,158.950
C06737=1022.071,-81.455,406.391,166.216,49.517,158.950
C06738=1022.066,-81.705,406.401,166.213,49.521,158.950
C06739=1022.059,-81.955,406.411,166.210,49.525,158.951
C06740=1022.054,-82.205,406.421,166.207,49.529,158.951
C06741=1022.048,-82.454,406.430,166.204,49.533,158.951
C06742=1022.043,-82.704,406.441,166.200,49.537,158.951
C06743=1022.037,-82.953,406.450,166.198,49.541,158.951
C06744=1022.031,-83.204,406.460,166.195,49.545,158.952
C06745=1022.025,-83.453,406.470,166.192,49.549,158.952
C06746=1022.020,-83.703,406.480,166.188,49.552,158.952
C06747=1022.014,-83.953,406.489,166.185,49.556,158.952
C06748=1022.008,-84.203,406.500,166.183,49.560,158.952
C06749=1022.002,-84.453,406.509,166.179,49.564,158.953
C06750=1021.997,-84.703,406.519,166.176,49.568,158.953
C06751=1021.990,-84.985,406.531,166.173,49.572,158.953
C06752=1021.984,-85.268,406.541,166.169,49.577,158.953
C06753=1021.977,-85.550,406.553,166.166,49.581,158.953
C06754=1021.971,-85.833,406.563,166.162,49.586,158.954
C06755=1021.966,-86.083,406.573,166.159,49.590,158.954
C06756=1021.960,-86.333,406.583,166.156,49.593,158.954
C06757=1021.955,-86.582,406.593,166.153,49.597,158.954
C06758=1021.949,-86.832,406.602,166.151,49.601,158.955
C06759=1021.943,-87.082,406.612,166.148,49.605,158.955
C06760=1021.937,-87.332,406.622,166.144,49.609,158.955
C06761=1021.931,-87.581,406.631,166.141,49.613,158.955
C06762=1021.926,-87.831,406.641,166.138,49.617,158.955
C06763=1021.920,-88.081,406.651,166.135,49.620,158.955
C06764=1021.915,-88.330,406.661,166.132,49.624,158.956
C06765=1021.909,-88.580,406.670,166.129,49.629,158.956
C06766=1021.903,-88.830,406.680,166.125,49.632,158.956
C06767=1021.898,-89.079,406.690,166.123,49.636,158.956
C06768=1021.892,-89.330,406.700,166.120,49.640,158.957
C06769=1021.886,-89.579,406.709,166.117,49.643,158.957
C06770=1021.881,-89.829,406.719,166.113,49.648,158.957
C06771=1021.875,-90.079,406.729,166.110,49.652,158.957
C06772=1021.870,-90.329,406.739,166.107,49.655,158.957
C06773=1021.864,-90.578,406.748,166.104,49.659,158.957
C06774=1021.858,-90.828,406.758,166.102,49.663,158.958
C06775=1021.853,-91.078,406.767,166.099,49.666,158.958
C06776=1021.847,-91.327,406.776,166.095,49.671,158.958
C06777=1021.842,-91.577,406.786,166.092,49.674,158.958
C06778=1021.836,-91.827,406.796,166.089,49.678,158.958
C06779=1021.831,-92.077,406.806,166.086,49.682,158.959
C06780=1021.825,-92.326,406.815,166.083,49.686,158.959
C06781=1021.820,-92.577,406.824,166.080,49.690,158.959
C06782=1021.814,-92.826,406.834,166.077,49.694,158.959
C06783=1021.809,-93.076,406.844,166.073,49.697,158.959
C06784=1021.803,-93.326,406.853,166.071,49.701,158.959
C06785=1021.797,-93.575,406.863,166.068,49.705,158.960
C06786=1021.792,-93.825,406.872,166.065,49.709,158.960
C06787=1021.787,-94.074,406.881,166.062,49.713,158.960
C06788=1021.781,-94.325,406.891,166.058,49.716,158.960
C06789=1021.776,-94.574,406.901,166.055,49.720,158.960
C06790=1021.770,-94.824,406.911,166.052,49.724,158.960
C06791=1021.765,-95.073,406.919,166.049,49.728,158.961
C06792=1021.759,-95.323,406.929,166.047,49.732,158.961
C06793=1021.754,-95.573,406.939,166.044,49.735,158.961
C06794=1021.748,-95.823,406.947,166.041,49.739,158.961
C06795=1021.743,-96.072,406.957,166.037,49.743,158.961
C06796=1021.737,-96.322,406.967,166.034,49.747,158.962
C06797=1021.732,-96.572,406.977,166.031,49.750,158.962
C06798=1021.726,-96.822,406.985,166.028,49.754,158.962
C06799=1021.721,-97.071,406.995,166.025,49.758,158.962
C06800=1021.716,-97.322,407.004,166.022,49.762,158.962
C06801=1021.710,-97.571,407.013,166.020,49.766,158.962
C06802=1021.705,-97.821,407.024,166.015,49.769,158.962
C06803=1021.699,-98.071,407.032,166.013,49.774,158.963
C06804=1021.693,-98.321,407.042,166.010,49.778,158.963
C06805=1021.688,-98.570,407.050,166.007,49.781,158.963
C06806=1021.682,-98.820,407.060,166.004,49.785,158.963
C06807=1021.677,-99.070,407.069,166.000,49.789,158.963
C06808=1021.671,-99.320,407.078,165.998,49.793,158.964
C06809=1021.666,-99.570,407.087,165.994,49.797,158.964
C06810=1021.660,-99.820,407.096,165.992,49.801,158.964
C06811=1021.654,-100.069,407.105,165.988,49.805,158.964
C06812=1021.649,-100.318,407.114,165.985,49.809,158.964
C06813=1021.643,-100.569,407.123,165.982,49.813,158.965
C06814=1021.638,-100.818,407.133,165.979,49.817,158.965
C06815=1021.633,-101.080,407.142,165.976,49.821,158.965
C06816=1021.627,-101.342,407.151,165.973,49.825,158.965
C06817=1021.620,-101.603,407.161,165.970,49.828,158.965
C06818=1021.614,-101.865,407.170,165.966,49.833,158.966
C06819=1021.610,-102.114,407.180,165.963,49.837,158.966
C06820=1021.604,-102.365,407.188,165.960,49.841,158.966
C06821=1021.598,-102.615,407.197,165.956,49.845,158.966
C06822=1021.593,-102.864,407.206,165.954,49.849,158.966
C06823=1021.587,-103.114,407.215,165.951,49.853,158.967
C06824=1021.582,-103.364,407.223,165.948,49.856,158.967
C06825=1021.576,-103.613,407.233,165.945,49.860,158.967
C06826=1021.571,-103.864,407.242,165.941,49.865,158.967
C06827=1021.566,-104.113,407.251,165.938,49.868,158.967
C06828=1021.560,-104.362,407.260,165.935,49.872,158.967
C06829=1021.554,-104.613,407.269,165.933,49.876,158.968
C06830=1021.549,-104.863,407.277,165.930,49.880,158.968
C06831=1021.543,-105.112,407.286,165.926,49.884,158.968
C06832=1021.538,-105.362,407.295,165.923,49.888,158.968
C06833=1021.532,-105.612,407.304,165.920,49.892,158.968
C06834=1021.527,-105.861,407.313,165.917,49.895,158.968
C06835=1021.521,-106.111,407.322,165.915,49.899,158.969
C06836=1021.516,-106.361,407.331,165.911,49.904,158.969
C06837=1021.511,-106.611,407.339,165.908,49.907,158.969
C06838=1021.506,-106.860,407.348,165.905,49.911,158.969
C06839=1021.500,-107.111,407.357,165.902,49.915,158.969
C06840=1021.494,-107.360,407.366,165.899,49.919,158.970
C06841=1021.489,-107.610,407.374,165.895,49.923,158.970
C06842=1021.483,-107.860,407.383,165.893,49.927,158.970
C06843=1021.478,-108.110,407.392,165.889,49.930,158.970
C06844=1021.472,-108.359,407.401,165.887,49.934,158.970
C06845=1021.467,-108.609,407.409,165.883,49.939,158.970
C06846=1021.462,-108.859,407.418,165.880,49.943,158.971
C06847=1021.455,-109.109,407.426,165.877,49.946,158.971
C06848=1021.450,-109.358,407.435,165.874,49.950,158.971
C06849=1021.445,-109.608,407.443,165.872,49.954,158.971
C06850=1021.440,-109.858,407.451,165.868,49.959,158.971
C06851=1021.434,-110.108,407.460,165.865,49.962,158.972
C06852=1021.428,-110.358,407.469,165.862,49.966,158.972
C06853=1021.423,-110.608,407.477,165.859,49.970,158.972
C06854=1021.418,-110.857,407.486,165.855,49.974,158.972
C06855=1021.413,-111.107,407.494,165.852,49.978,158.972
C06856=1021.406,-111.357,407.504,165.850,49.982,158.973
C06857=1021.401,-111.607,407.512,165.847,49.986,158.973
C06858=1021.396,-111.856,407.521,165.844,49.990,158.973
C06859=1021.390,-112.106,407.529,165.840,49.994,158.973
C06860=1021.385,-112.356,407.537,165.837,49.998,158.973
C06861=1021.379,-112.605,407.546,165.834,50.001,158.973
C06862=1021.374,-112.855,407.554,165.832,50.005,158.974
C06863=1021.368,-113.105,407.563,165.828,50.010,158.974
C06864=1021.363,-113.356,407.571,165.825,50.013,158.974
C06865=1021.358,-113.605,407.579,165.822,50.017,158.974
C06866=1021.353,-113.855,407.588,165.819,50.021,158.974
C06867=1021.347,-114.128,407.597,165.816,50.026,158.974
C06868=1021.341,-114.400,407.606,165.813,50.030,158.975
C06869=1021.335,-114.674,407.616,165.809,50.034,158.975
C06870=1021.329,-114.947,407.625,165.805,50.039,158.975
C06871=1021.324,-115.197,407.633,165.803,50.043,158.975
C06872=1021.319,-115.447,407.641,165.800,50.047,158.975
C06873=1021.313,-115.696,407.649,165.797,50.050,158.976
C06874=1021.307,-115.946,407.658,165.793,50.055,158.976
C06875=1021.302,-116.196,407.666,165.790,50.059,158.976
C06876=1021.297,-116.445,407.675,165.787,50.062,158.976
C06877=1021.291,-116.695,407.682,165.784,50.066,158.976
C06878=1021.286,-116.945,407.690,165.782,50.070,158.977
C06879=1021.279,-117.230,407.700,165.778,50.075,158.977
C06880=1021.273,-117.515,407.709,165.774,50.079,158.977
C06881=1021.267,-117.800,407.719,165.771,50.084,158.977
C06882=1021.261,-118.085,407.728,165.767,50.089,158.977
C06883=1021.255,-118.334,407.737,165.764,50.093,158.977
C06884=1021.250,-118.584,407.744,165.761,50.096,158.978
C06885=1021.245,-118.834,407.752,165.758,50.100,158.978
C06886=1021.239,-119.084,407.761,165.755,50.105,158.978
C06887=1021.234,-119.333,407.769,165.752,50.109,158.978
C06888=1021.228,-119.584,407.777,165.749,50.112,158.978
C06889=1021.223,-119.833,407.785,165.746,50.116,158.979
C06890=1021.218,-120.083,407.794,165.743,50.120,158.979
C06891=1021.212,-120.333,407.801,165.740,50.125,158.979
C06892=1021.207,-120.583,407.809,165.737,50.128,158.979
C06893=1021.202,-120.832,407.818,165.734,50.132,158.979
C06894=1021.196,-121.082,407.825,165.731,50.136,158.979
C06895=1021.191,-121.331,407.833,165.727,50.140,158.979
C06896=1021.186,-121.581,407.842,165.724,50.144,158.980
C06897=1021.181,-121.831,407.849,165.722,50.148,158.980
C06898=1021.175,-122.081,407.857,165.719,50.152,158.980
C06899=1021.170,-122.331,407.865,165.716,50.156,158.980
C06900=1021.165,-122.581,407.873,165.712,50.160,158.980
C06901=1021.159,-122.830,407.881,165.709,50.164,158.981
C06902=1021.154,-123.081,407.889,165.706,50.167,158.981
C06903=1021.149,-123.330,407.898,165.703,50.171,158.981
C06904=1021.143,-123.580,407.905,165.701,50.176,158.981
C06905=1021.138,-123.830,407.913,165.697,50.180,158.981
C06906=1021.133,-124.080,407.921,165.694,50.183,158.981
C06907=1021.127,-124.329,407.929,165.691,50.187,158.982
C06908=1021.122,-124.579,407.936,165.688,50.192,158.982
C06909=1021.116,-124.829,407.944,165.684,50.195,158.982
C06910=1021.111,-125.079,407.952,165.682,50.199,158.982
C06911=1021.105,-125.329,407.960,165.679,50.203,158.982
C06912=1021.100,-125.579,407.968,165.676,50.208,158.983
C06913=1021.095,-125.829,407.976,165.672,50.212,158.983
///RCONF 1,0,0,0,1,0,0,0,0,0,0,0,0,0,0,0,0,0,0,0,0,0,0,0
C06914=1021.089,-126.079,407.983,165.669,50.215,158.983
C06915=1021.085,-126.328,407.991,165.667,50.220,158.983
C06916=1021.079,-126.578,407.999,165.664,50.224,158.983
C06917=1021.074,-126.828,408.006,165.661,50.228,158.984
C06918=1021.068,-127.077,408.014,165.657,50.231,158.983
C06919=1021.063,-127.328,408.022,165.654,50.236,158.984
C06920=1021.058,-127.577,408.030,165.652,50.240,158.984
C06921=1021.053,-127.827,408.037,165.649,50.244,158.984
C06922=1021.047,-128.077,408.044,165.645,50.247,158.984
C06923=1021.042,-128.326,408.053,165.643,50.251,158.984
C06924=1021.038,-128.575,408.062,165.640,50.254,158.984
C06925=1021.034,-128.825,408.072,165.637,50.256,158.984
C06926=1021.031,-129.075,408.081,165.633,50.258,158.984
C06927=1021.028,-129.325,408.092,165.632,50.260,158.984
C06928=1021.026,-129.574,408.103,165.629,50.260,158.984
C06929=1021.023,-129.824,408.115,165.626,50.261,158.983
C06930=1021.022,-130.074,408.127,165.624,50.261,158.983
C06931=1021.021,-130.324,408.140,165.621,50.260,158.982
C06932=1021.021,-130.574,408.154,165.619,50.259,158.982
C06933=1021.020,-130.823,408.169,165.617,50.257,158.981
C06934=1021.021,-131.073,408.183,165.615,50.255,158.981
C06935=1021.021,-131.323,408.198,165.613,50.253,158.980
C06936=1021.023,-131.572,408.215,165.611,50.250,158.979
C06937=1021.025,-131.822,408.231,165.609,50.245,158.978
C06938=1021.027,-132.072,408.248,165.607,50.242,158.977
C06939=1021.030,-132.322,408.266,165.606,50.236,158.976
C06940=1021.033,-132.571,408.283,165.604,50.232,158.975
C06941=1021.037,-132.821,408.303,165.603,50.226,158.973
C06942=1021.040,-133.071,408.322,165.601,50.220,158.972
C06943=1020.759,-133.097,407.965,165.556,50.526,159.017
C06944=1020.755,-132.847,407.946,165.556,50.532,159.018
C06945=1020.752,-132.597,407.927,165.558,50.538,159.019
C06946=1020.748,-132.348,407.909,165.560,50.543,159.020
C06947=1020.746,-132.098,407.891,165.562,50.547,159.021
C06948=1020.743,-131.849,407.874,165.563,50.552,159.022
C06949=1020.741,-131.598,407.858,165.565,50.556,159.023
C06950=1020.741,-131.349,407.842,165.568,50.559,159.024
C06951=1020.739,-131.098,407.827,165.569,50.561,159.025
C06952=1020.739,-130.849,407.812,165.571,50.564,159.026
C06953=1020.739,-130.599,407.797,165.574,50.566,159.026
C06954=1020.740,-130.349,407.784,165.576,50.566,159.027
C06955=1020.741,-130.100,407.771,165.578,50.567,159.027
C06956=1020.742,-129.850,407.759,165.580,50.567,159.028
C06957=1020.744,-129.601,407.747,165.584,50.567,159.028
C06958=1020.747,-129.350,407.735,165.585,50.565,159.028
C06959=1020.749,-129.101,407.724,165.589,50.564,159.029
C06960=1020.753,-128.851,407.715,165.591,50.562,159.029
C06961=1020.756,-128.601,407.705,165.593,50.560,159.029
C06962=1020.761,-128.352,407.696,165.597,50.557,159.029
C06963=1020.766,-128.102,407.688,165.600,50.554,159.029
C06964=1020.771,-127.853,407.681,165.603,50.549,159.029
C06965=1020.776,-127.603,407.673,165.605,50.545,159.028
C06966=1020.782,-127.354,407.665,165.609,50.541,159.028
C06967=1020.787,-127.103,407.657,165.612,50.537,159.028
C06968=1020.792,-126.855,407.650,165.615,50.533,159.028
C06969=1020.797,-126.604,407.642,165.617,50.529,159.028
C06970=1020.803,-126.354,407.635,165.621,50.525,159.028
C06971=1020.808,-126.105,407.626,165.624,50.521,159.027
C06972=1020.813,-125.854,407.619,165.627,50.517,159.027
C06973=1020.819,-125.606,407.611,165.631,50.513,159.027
C06974=1020.823,-125.355,407.603,165.633,50.509,159.027
C06975=1020.829,-125.105,407.596,165.636,50.504,159.027
C06976=1020.834,-124.855,407.588,165.639,50.500,159.026
C06977=1020.840,-124.605,407.580,165.642,50.496,159.026
C06978=1020.845,-124.356,407.572,165.646,50.492,159.026
C06979=1020.851,-124.106,407.565,165.648,50.488,159.026
///RCONF 1,0,0,0,0,0,0,0,0,0,0,0,0,0,0,0,0,0,0,0,0,0,0,0
C06980=1020.856,-123.857,407.557,165.651,50.484,159.026
C06981=1020.861,-123.606,407.549,165.655,50.481,159.026
C06982=1020.867,-123.357,407.541,165.658,50.476,159.025
C06983=1020.872,-123.107,407.533,165.660,50.472,159.025
C06984=1020.877,-122.857,407.525,165.663,50.468,159.025
C06985=1020.883,-122.607,407.518,165.667,50.464,159.025
C06986=1020.888,-122.357,407.509,165.670,50.460,159.025
C06987=1020.893,-122.107,407.501,165.673,50.456,159.025
C06988=1020.899,-121.857,407.493,165.675,50.452,159.024
C06989=1020.904,-121.608,407.485,165.679,50.448,159.024
C06990=1020.908,-121.358,407.478,165.682,50.444,159.024
C06991=1020.914,-121.109,407.470,165.685,50.440,159.024
C06992=1020.920,-120.859,407.461,165.688,50.436,159.024
C06993=1020.925,-120.609,407.453,165.691,50.431,159.023
C06994=1020.930,-120.359,407.445,165.694,50.428,159.023
C06995=1020.936,-120.109,407.438,165.697,50.424,159.023
C06996=1020.941,-119.859,407.429,165.700,50.420,159.023
C06997=1020.946,-119.609,407.421,165.703,50.415,159.023
C06998=1020.952,-119.359,407.414,165.707,50.412,159.023
C06999=1020.957,-119.110,407.405,165.709,50.408,159.022
C07000=1020.962,-118.860,407.397,165.712,50.404,159.022
C07001=1020.967,-118.610,407.389,165.716,50.399,159.022
C07002=1020.973,-118.360,407.381,165.718,50.395,159.022
C07003=1020.979,-118.111,407.373,165.721,50.392,159.022
C07004=1020.985,-117.826,407.363,165.725,50.387,159.021
C07005=1020.991,-117.542,407.354,165.729,50.382,159.021
C07006=1020.997,-117.257,407.344,165.732,50.378,159.021
C07007=1021.003,-116.972,407.335,165.736,50.373,159.021
C07008=1021.009,-116.722,407.328,165.739,50.369,159.021
C07009=1021.014,-116.472,407.319,165.741,50.365,159.021
C07010=1021.019,-116.222,407.311,165.744,50.361,159.020
C07011=1021.025,-115.973,407.302,165.748,50.357,159.020
C07012=1021.031,-115.723,407.294,165.751,50.352,159.020
C07013=1021.036,-115.473,407.286,165.754,50.349,159.020
C07014=1021.041,-115.223,407.278,165.757,50.345,159.020
C07015=1021.046,-114.973,407.269,165.760,50.341,159.019
C07016=1021.051,-114.724,407.261,165.763,50.336,159.019
C07017=1021.057,-114.474,407.253,165.765,50.332,159.019
C07018=1021.063,-114.225,407.245,165.770,50.329,159.019
C07019=1021.068,-113.975,407.236,165.772,50.325,159.019
C07020=1021.073,-113.724,407.228,165.775,50.320,159.018
C07021=1021.079,-113.474,407.219,165.778,50.317,159.018
C07022=1021.084,-113.224,407.211,165.782,50.313,159.018
C07023=1021.089,-112.975,407.203,165.785,50.308,159.018
C07024=1021.094,-112.725,407.194,165.787,50.304,159.018
C07025=1021.100,-112.475,407.186,165.790,50.301,159.018
C07026=1021.105,-112.226,407.177,165.794,50.297,159.018
C07027=1021.111,-111.976,407.169,165.797,50.292,159.017
C07028=1021.117,-111.726,407.160,165.799,50.288,159.017
C07029=1021.122,-111.476,407.152,165.803,50.285,159.017
C07030=1021.127,-111.226,407.143,165.806,50.281,159.017
C07031=1021.133,-110.977,407.135,165.809,50.276,159.017
C07032=1021.138,-110.727,407.126,165.812,50.272,159.016
C07033=1021.143,-110.477,407.118,165.815,50.269,159.016
C07034=1021.148,-110.227,407.109,165.819,50.265,159.016
C07035=1021.154,-109.977,407.101,165.821,50.260,159.016
C07036=1021.160,-109.727,407.092,165.824,50.256,159.016
C07037=1021.165,-109.478,407.084,165.827,50.252,159.015
C07038=1021.170,-109.228,407.075,165.831,50.248,159.015
C07039=1021.176,-108.979,407.067,165.833,50.244,159.015
C07040=1021.182,-108.729,407.058,165.836,50.240,159.015
C07041=1021.188,-108.479,407.049,165.840,50.236,159.015
C07042=1021.193,-108.229,407.041,165.843,50.232,159.014
C07043=1021.198,-107.980,407.032,165.846,50.228,159.014
C07044=1021.204,-107.729,407.023,165.848,50.224,159.014
C07045=1021.209,-107.479,407.015,165.852,50.220,159.014
C07046=1021.214,-107.230,407.006,165.855,50.216,159.014
C07047=1021.220,-106.981,406.997,165.858,50.212,159.014
C07048=1021.226,-106.730,406.988,165.861,50.208,159.013
C07049=1021.231,-106.480,406.980,165.864,50.204,159.013
C07050=1021.236,-106.231,406.971,165.867,50.200,159.013
C07051=1021.241,-105.981,406.962,165.870,50.196,159.013
C07052=1021.247,-105.731,406.953,165.873,50.192,159.013
C07053=1021.252,-105.481,406.944,165.877,50.188,159.012
C07054=1021.258,-105.231,406.936,165.880,50.185,159.012
C07055=1021.263,-104.982,406.927,165.882,50.180,159.012
C07056=1021.269,-104.732,406.918,165.885,50.176,159.012
C07057=1021.274,-104.482,406.909,165.889,50.172,159.012
C07058=1021.280,-104.233,406.901,165.892,50.169,159.012
C07059=1021.286,-103.983,406.891,165.895,50.164,159.011
C07060=1021.291,-103.733,406.883,165.897,50.160,159.011
C07061=1021.296,-103.483,406.874,165.901,50.156,159.011
C07062=1021.301,-103.233,406.865,165.904,50.153,159.011
C07063=1021.307,-102.983,406.856,165.907,50.148,159.011
C07064=1021.312,-102.734,406.847,165.910,50.144,159.010
C07065=1021.318,-102.484,406.837,165.913,50.140,159.010
C07066=1021.324,-102.234,406.829,165.916,50.137,159.010
C07067=1021.329,-101.985,406.821,165.919,50.133,159.010
C07068=1021.335,-101.700,406.810,165.923,50.128,159.010
C07069=1021.342,-101.414,406.800,165.926,50.123,159.009
C07070=1021.347,-101.130,406.789,165.930,50.119,159.009
C07071=1021.354,-100.845,406.779,165.933,50.115,159.009
C07072=1021.360,-100.546,406.769,165.937,50.109,159.009
C07073=1021.367,-100.246,406.758,165.941,50.105,159.009
C07074=1021.374,-99.946,406.747,165.944,50.100,159.008
C07075=1021.381,-99.647,406.736,165.948,50.095,159.008
C07076=1021.386,-99.397,406.727,165.951,50.091,159.008
C07077=1021.391,-99.148,406.717,165.954,50.087,159.008
C07078=1021.397,-98.898,406.709,165.957,50.083,159.008
C07079=1021.403,-98.648,406.699,165.960,50.079,159.007
C07080=1021.408,-98.398,406.690,165.963,50.075,159.007
C07081=1021.414,-98.149,406.681,165.967,50.071,159.007
C07082=1021.420,-97.898,406.672,165.970,50.067,159.007
C07083=1021.425,-97.649,406.663,165.972,50.063,159.007
C07084=1021.431,-97.399,406.654,165.975,50.059,159.006
C07085=1021.435,-97.149,406.644,165.978,50.055,159.006
C07086=1021.441,-96.900,406.635,165.982,50.052,159.006
C07087=1021.447,-96.650,406.626,165.985,50.047,159.006
C07088=1021.452,-96.400,406.616,165.988,50.043,159.006
C07089=1021.458,-96.151,406.607,165.991,50.040,159.006
C07090=1021.462,-95.901,406.598,165.993,50.036,159.005
C07091=1021.469,-95.651,406.588,165.998,50.032,159.005
C07092=1021.473,-95.401,406.578,166.000,50.028,159.005
C07093=1021.480,-95.152,406.569,166.003,50.024,159.005
C07094=1021.485,-94.902,406.560,166.006,50.021,159.005
C07095=1021.490,-94.652,406.550,166.009,50.017,159.004
C07096=1021.496,-94.403,406.541,166.011,50.013,159.004
C07097=1021.501,-94.152,406.531,166.016,50.009,159.004
C07098=1021.507,-93.903,406.522,166.018,50.005,159.004
C07099=1021.512,-93.653,406.512,166.021,50.001,159.004
C07100=1021.518,-93.404,406.503,166.024,49.997,159.004
C07101=1021.523,-93.153,406.494,166.028,49.993,159.003
C07102=1021.528,-92.904,406.484,166.031,49.989,159.003
C07103=1021.534,-92.654,406.475,166.034,49.986,159.003
C07104=1021.540,-92.404,406.464,166.036,49.981,159.003
C07105=1021.545,-92.155,406.455,166.039,49.977,159.003
C07106=1021.551,-91.904,406.446,166.043,49.974,159.003
C07107=1021.556,-91.655,406.437,166.046,49.970,159.002
C07108=1021.562,-91.405,406.426,166.049,49.966,159.002
C07109=1021.567,-91.156,406.417,166.051,49.962,159.002
C07110=1021.573,-90.906,406.408,166.055,49.958,159.002
C07111=1021.579,-90.656,406.397,166.058,49.954,159.002
C07112=1021.584,-90.406,406.389,166.061,49.950,159.001
C07113=1021.589,-90.156,406.379,166.064,49.946,159.001
C07114=1021.595,-89.907,406.370,166.067,49.942,159.001
C07115=1021.600,-89.657,406.359,166.071,49.938,159.001
C07116=1021.607,-89.407,406.350,166.073,49.934,159.001
C07117=1021.611,-89.158,406.340,166.076,49.930,159.000
C07118=1021.618,-88.908,406.330,166.079,49.926,159.000
C07119=1021.623,-88.658,406.320,166.082,49.922,159.000
C07120=1021.629,-88.409,406.311,166.086,49.919,159.000
C07121=1021.634,-88.158,406.302,166.089,49.915,159.000
C07122=1021.640,-87.908,406.292,166.091,49.911,158.999
C07123=1021.645,-87.659,406.283,166.094,49.906,158.999
C07124=1021.651,-87.409,406.273,166.098,49.903,158.999
C07125=1021.657,-87.159,406.263,166.101,49.899,158.999
C07126=1021.662,-86.910,406.253,166.104,49.895,158.999
C07127=1021.668,-86.660,406.244,166.106,49.891,158.998
C07128=1021.673,-86.419,406.234,166.109,49.887,158.998
C07129=1021.679,-86.177,406.225,166.113,49.883,158.998
C07130=1021.684,-85.936,406.215,166.116,49.879,158.998
C07131=1021.690,-85.695,406.206,166.119,49.876,158.998
C07132=1021.696,-85.453,406.196,166.122,49.871,158.997
C07133=1021.701,-85.212,406.187,166.125,49.867,158.997
C07134=1021.706,-84.970,406.177,166.128,49.864,158.997
C07135=1021.711,-84.729,406.168,166.130,49.860,158.997
C07136=1021.717,-84.479,406.158,166.133,49.856,158.997
C07137=1021.723,-84.229,406.149,166.137,49.852,158.996
C07138=1021.728,-83.980,406.139,166.140,49.848,158.996
C07139=1021.735,-83.730,406.129,166.143,49.844,158.996
C07140=1021.740,-83.480,406.119,166.145,49.840,158.996
C07141=1021.746,-83.230,406.110,166.149,49.836,158.996
C07142=1021.751,-82.981,406.099,166.152,49.832,158.995
C07143=1021.757,-82.732,406.090,166.155,49.828,158.995
C07144=1021.763,-82.482,406.079,166.158,49.824,158.995
C07145=1021.769,-82.232,406.070,166.161,49.820,158.995
C07146=1021.774,-81.982,406.060,166.164,49.816,158.994
C07147=1021.780,-81.733,406.050,166.167,49.812,158.994
C07148=1021.785,-81.482,406.040,166.170,49.808,158.994
C07149=1021.792,-81.233,406.031,166.173,49.803,158.994
C07150=1021.797,-80.983,406.020,166.177,49.800,158.994
C07151=1021.804,-80.733,406.010,166.179,49.796,158.993
C07152=1021.809,-80.483,406.000,166.183,49.792,158.993
C07153=1021.815,-80.234,405.991,166.186,49.788,158.993
C07154=1021.820,-79.984,405.981,166.188,49.784,158.993
C07155=1021.826,-79.735,405.970,166.192,49.780,158.993
C07156=1021.831,-79.484,405.960,166.194,49.776,158.992
C07157=1021.837,-79.235,405.950,166.198,49.772,158.992
C07158=1021.843,-78.985,405.939,166.201,49.768,158.992
C07159=1021.848,-78.735,405.929,166.204,49.764,158.992
C07160=1021.853,-78.486,405.919,166.207,49.760,158.992
C07161=1021.860,-78.236,405.909,166.210,49.757,158.991
C07162=1021.865,-77.986,405.899,166.212,49.753,158.991
C07163=1021.871,-77.736,405.889,166.216,49.749,158.991
C07164=1021.876,-77.487,405.878,166.219,49.745,158.991
C07165=1021.882,-77.237,405.868,166.222,49.741,158.991
C07166=1021.888,-76.987,405.858,166.225,49.737,158.990
C07167=1021.894,-76.737,405.847,166.227,49.733,158.990
C07168=1021.899,-76.488,405.837,166.232,49.729,158.990
C07169=1021.904,-76.238,405.827,166.234,49.725,158.990
C07170=1021.911,-75.989,405.817,166.237,49.721,158.989
C07171=1021.916,-75.739,405.806,166.240,49.717,158.989
C07172=1021.922,-75.489,405.796,166.243,49.714,158.989
C07173=1021.927,-75.239,405.786,166.247,49.710,158.989
C07174=1021.933,-74.989,405.775,166.249,49.706,158.989
C07175=1021.939,-74.740,405.765,166.252,49.702,158.988
C07176=1021.945,-74.490,405.754,166.255,49.698,158.988
C07177=1021.950,-74.240,405.744,166.258,49.694,158.988
C07178=1021.956,-73.991,405.733,166.261,49.690,158.988
C07179=1021.961,-73.740,405.723,166.265,49.687,158.988
C07180=1021.967,-73.491,405.712,166.268,49.682,158.987
C07181=1021.973,-73.241,405.701,166.271,49.679,158.987
C07182=1021.978,-72.991,405.691,166.273,49.675,158.987
C07183=1021.984,-72.742,405.680,166.277,49.672,158.987
C07184=1021.989,-72.492,405.669,166.279,49.668,158.987
C07185=1021.994,-72.242,405.659,166.282,49.664,158.987
C07186=1022.000,-71.992,405.648,166.285,49.660,158.986
C07187=1022.006,-71.743,405.637,166.288,49.656,158.986
C07188=1022.011,-71.493,405.627,166.291,49.653,158.986
C07189=1022.017,-71.243,405.616,166.295,49.649,158.986
C07190=1022.023,-70.994,405.605,166.298,49.645,158.986
C07191=1022.028,-70.744,405.595,166.301,49.641,158.985
C07192=1022.034,-70.494,405.584,166.303,49.637,158.985
C07193=1022.040,-70.245,405.573,166.306,49.634,158.985
C07194=1022.045,-69.995,405.562,166.309,49.630,158.985
C07195=1022.051,-69.745,405.552,166.312,49.627,158.985
C07196=1022.057,-69.465,405.539,166.316,49.622,158.984
C07197=1022.063,-69.184,405.528,166.319,49.618,158.984
C07198=1022.070,-68.903,405.515,166.322,49.613,158.984
C07199=1022.076,-68.622,405.503,166.326,49.609,158.984
C07200=1022.082,-68.373,405.493,166.329,49.606,158.984
C07201=1022.087,-68.123,405.482,166.332,49.601,158.983
C07202=1022.093,-67.874,405.471,166.335,49.598,158.983
C07203=1022.099,-67.624,405.460,166.338,49.594,158.983
C07204=1022.104,-67.374,405.450,166.340,49.590,158.983
C07205=1022.110,-67.125,405.439,166.343,49.587,158.983
C07206=1022.115,-66.875,405.427,166.347,49.582,158.982
C07207=1022.121,-66.626,405.417,166.350,49.578,158.982
C07208=1022.127,-66.376,405.406,166.353,49.575,158.982
C07209=1022.132,-66.127,405.395,166.356,49.571,158.982
C07210=1022.138,-65.876,405.384,166.359,49.567,158.981
C07211=1022.144,-65.626,405.373,166.362,49.564,158.981
C07212=1022.150,-65.377,405.363,166.364,49.560,158.981
C07213=1022.156,-65.127,405.352,166.368,49.555,158.981
C07214=1022.161,-64.878,405.341,166.371,49.552,158.981
C07215=1022.166,-64.628,405.329,166.374,49.548,158.980
C07216=1022.172,-64.378,405.318,166.377,49.544,158.980
C07217=1022.178,-64.128,405.307,166.379,49.540,158.980
C07218=1022.184,-63.879,405.296,166.383,49.537,158.980
C07219=1022.190,-63.629,405.286,166.385,49.533,158.979
C07220=1022.195,-63.379,405.275,166.388,49.529,158.979
C07221=1022.201,-63.130,405.264,166.392,49.525,158.979
C07222=1022.207,-62.880,405.254,166.395,49.521,158.979
C07223=1022.213,-62.630,405.242,166.398,49.517,158.979
C07224=1022.218,-62.380,405.231,166.400,49.513,158.978
C07225=1022.224,-62.131,405.220,166.404,49.510,158.978
C07226=1022.230,-61.881,405.209,166.406,49.506,158.978
C07227=1022.236,-61.631,405.198,166.409,49.502,158.978
C07228=1022.242,-61.382,405.187,166.413,49.498,158.978
C07229=1022.247,-61.132,405.176,166.416,49.494,158.977
C07230=1022.253,-60.883,405.165,166.419,49.490,158.977
C07231=1022.259,-60.633,405.154,166.421,49.486,158.977
C07232=1022.264,-60.383,405.142,166.424,49.482,158.977
C07233=1022.270,-60.133,405.132,166.427,49.479,158.976
C07234=1022.276,-59.884,405.121,166.431,49.474,158.976
C07235=1022.282,-59.634,405.110,166.434,49.470,158.976
C07236=1022.288,-59.385,405.098,166.437,49.466,158.976
C07237=1022.294,-59.135,405.087,166.440,49.463,158.976
C07238=1022.300,-58.886,405.076,166.442,49.459,158.975
C07239=1022.305,-58.635,405.064,166.445,49.455,158.975
C07240=1022.311,-58.386,405.053,166.448,49.451,158.975
C07241=1022.317,-58.136,405.043,166.452,49.447,158.975
C07242=1022.323,-57.887,405.032,166.455,49.443,158.974
C07243=1022.329,-57.636,405.020,166.458,49.439,158.974
C07244=1022.335,-57.387,405.010,166.460,49.435,158.974
C07245=1022.340,-57.137,404.999,166.463,49.431,158.974
C07246=1022.346,-56.888,404.986,166.466,49.427,158.973
C07247=1022.352,-56.638,404.975,166.470,49.424,158.973
C07248=1022.358,-56.389,404.964,166.473,49.420,158.973
C07249=1022.364,-56.138,404.953,166.475,49.416,158.973
C07250=1022.370,-55.889,404.942,166.478,49.412,158.972
C07251=1022.376,-55.639,404.931,166.481,49.408,158.972
C07252=1022.382,-55.390,404.919,166.484,49.404,158.972
C07253=1022.387,-55.140,404.908,166.488,49.400,158.972
C07254=1022.394,-54.890,404.897,166.491,49.396,158.971
C07255=1022.399,-54.640,404.886,166.493,49.392,158.971
C07256=1022.405,-54.391,404.875,166.496,49.388,158.971
C07257=1022.412,-54.141,404.863,166.499,49.384,158.971
C07258=1022.418,-53.892,404.852,166.502,49.380,158.970
C07259=1022.423,-53.641,404.840,166.505,49.376,158.970
C07260=1022.430,-53.363,404.828,166.508,49.372,158.970
C07261=1022.437,-53.083,404.815,166.512,49.367,158.970
C07262=1022.443,-52.803,404.803,166.515,49.362,158.969
C07263=1022.450,-52.524,404.790,166.518,49.358,158.969
C07264=1022.456,-52.274,404.779,166.521,49.354,158.969
C07265=1022.462,-52.025,404.767,166.525,49.350,158.969
C07266=1022.467,-51.775,404.756,166.527,49.346,158.968
C07267=1022.474,-51.525,404.744,166.530,49.342,158.968
C07268=1022.480,-51.276,404.733,166.533,49.338,158.968
C07269=1022.485,-51.026,404.722,166.536,49.335,158.968
C07270=1022.492,-50.776,404.711,166.540,49.330,158.967
C07271=1022.497,-50.527,404.698,166.543,49.326,158.967
C07272=1022.503,-50.276,404.687,166.545,49.322,158.967
C07273=1022.509,-50.028,404.675,166.548,49.319,158.967
C07274=1022.514,-49.777,404.663,166.551,49.315,158.966
C07275=1022.520,-49.528,404.652,166.554,49.312,158.966
